// TIA Portal V17 export
// export: Created 2023-08-28T22:41:32.6164324Z, ExportSetting WithDefaults, DisplayName Totally Integrated Automation Portal, DisplayVersion V17 Update 5, DisplayName TIA Portal Openness, DisplayVersion V17 Update 5, DisplayName TIA Portal Teamcenter Gateway, DisplayVersion V17 Update 5, DisplayName TIA Portal Version Control Interface, DisplayVersion V17, DisplayName Simotion SCOUT TIA, DisplayVersion 5.4.3.0, DisplayName TIA Portal Test Suite Advanced, DisplayVersion V17 Update 1, DisplayName SIMOCODE ES, DisplayVersion V17 Update 5, DisplayName SINAMICS Startdrive Advanced, DisplayVersion V17 SP1, DisplayName SINAMICS Startdrive G130, G150, S120, S150, SINAMICS MV, S210, DisplayVersion V17 SP1, DisplayName SINAMICS Startdrive G110M, G120, G120C, G120D, G120P, G115D, DisplayVersion V17 SP1, DisplayName SIRIUS Safety ES, DisplayVersion V17 Update 5, DisplayName STEP 7 Professional, DisplayVersion V17 Update 5, DisplayName STEP 7 CFC, DisplayVersion V17 Update 1, DisplayName STEP 7 Safety, DisplayVersion V17, DisplayName WinCC Advanced, DisplayVersion V17 Update 5, DisplayName SIMATIC Visualization Architect, DisplayVersion V17 Update 5
DATA_BLOCK "S1.CABINET000.ALARM1"   // DB2200
// stored: AutoNumber true, DBAccessibleFromOPCUA true, DBAccessibleFromWebserver true, InstanceOfName BoolToUDInt_Inverted_Filtered, InstanceOfType FB
"BoolToUDInt_Inverted_Filtered "
BEGIN
END_DATA_BLOCK

DATA_BLOCK "S1.CABINET000.ALARM2"   // DB2201
// stored: AutoNumber true, DBAccessibleFromOPCUA true, DBAccessibleFromWebserver true, InstanceOfName BoolToUDInt_Inverted_Filtered, InstanceOfType FB
"BoolToUDInt_Inverted_Filtered "
BEGIN
END_DATA_BLOCK

DATA_BLOCK "S1.CABINET000.WARNING1"   // DB2202
// stored: AutoNumber true, DBAccessibleFromOPCUA true, DBAccessibleFromWebserver true, InstanceOfName BoolToUDInt_Inverted_Filtered, InstanceOfType FB
"BoolToUDInt_Inverted_Filtered "
BEGIN
END_DATA_BLOCK

DATA_BLOCK "S1.CABINET000.WARNING2"   // DB2203
// stored: AutoNumber true, DBAccessibleFromOPCUA true, DBAccessibleFromWebserver true, InstanceOfName BoolToUDInt_Inverted_Filtered, InstanceOfType FB
"BoolToUDInt_Inverted_Filtered "
BEGIN
END_DATA_BLOCK

DATA_BLOCK "S1.CABINET001.ALARM1"   // DB2204
// stored: AutoNumber true, DBAccessibleFromOPCUA true, DBAccessibleFromWebserver true, InstanceOfName BoolToUDInt_Inverted_Filtered, InstanceOfType FB
"BoolToUDInt_Inverted_Filtered "
BEGIN
END_DATA_BLOCK

DATA_BLOCK "S1.CABINET001.ALARM2"   // DB2205
// stored: AutoNumber true, DBAccessibleFromOPCUA true, DBAccessibleFromWebserver true, InstanceOfName BoolToUDInt_Inverted_Filtered, InstanceOfType FB
"BoolToUDInt_Inverted_Filtered "
BEGIN
END_DATA_BLOCK

DATA_BLOCK "S1.CABINET001.WARNING1"   // DB2206
// stored: AutoNumber true, DBAccessibleFromOPCUA true, DBAccessibleFromWebserver true, InstanceOfName BoolToUDInt_Inverted_Filtered, InstanceOfType FB
"BoolToUDInt_Inverted_Filtered "
BEGIN
END_DATA_BLOCK

DATA_BLOCK "S1.CABINET001.WARNING2"   // DB2207
// stored: AutoNumber true, DBAccessibleFromOPCUA true, DBAccessibleFromWebserver true, InstanceOfName BoolToUDInt_Inverted_Filtered, InstanceOfType FB
"BoolToUDInt_Inverted_Filtered "
BEGIN
END_DATA_BLOCK

DATA_BLOCK "S1.CABINET002.ALARM1"   // DB2208
// stored: AutoNumber true, DBAccessibleFromOPCUA true, DBAccessibleFromWebserver true, InstanceOfName BoolToUDInt_Inverted_Filtered, InstanceOfType FB
"BoolToUDInt_Inverted_Filtered "
BEGIN
END_DATA_BLOCK

DATA_BLOCK "S1.CABINET002.ALARM2"   // DB2209
// stored: AutoNumber true, DBAccessibleFromOPCUA true, DBAccessibleFromWebserver true, InstanceOfName BoolToUDInt_Inverted_Filtered, InstanceOfType FB
"BoolToUDInt_Inverted_Filtered "
BEGIN
END_DATA_BLOCK

DATA_BLOCK "S1.CABINET002.WARNING1"   // DB2210
// stored: AutoNumber true, DBAccessibleFromOPCUA true, DBAccessibleFromWebserver true, InstanceOfName BoolToUDInt_Inverted_Filtered, InstanceOfType FB
"BoolToUDInt_Inverted_Filtered "
BEGIN
END_DATA_BLOCK

DATA_BLOCK "S1.CABINET002.WARNING2"   // DB2211
// stored: AutoNumber true, DBAccessibleFromOPCUA true, DBAccessibleFromWebserver true, InstanceOfName BoolToUDInt_Inverted_Filtered, InstanceOfType FB
"BoolToUDInt_Inverted_Filtered "
BEGIN
END_DATA_BLOCK

DATA_BLOCK "S1.CABINET003.ALARM1"   // DB2212
// stored: AutoNumber true, DBAccessibleFromOPCUA true, DBAccessibleFromWebserver true, InstanceOfName BoolToUDInt_Inverted_Filtered, InstanceOfType FB
"BoolToUDInt_Inverted_Filtered "
BEGIN
END_DATA_BLOCK

DATA_BLOCK "S1.CABINET003.ALARM2"   // DB2213
// stored: AutoNumber true, DBAccessibleFromOPCUA true, DBAccessibleFromWebserver true, InstanceOfName BoolToUDInt_Inverted_Filtered, InstanceOfType FB
"BoolToUDInt_Inverted_Filtered "
BEGIN
END_DATA_BLOCK

DATA_BLOCK "S1.CABINET003.WARNING1"   // DB2214
// stored: AutoNumber true, DBAccessibleFromOPCUA true, DBAccessibleFromWebserver true, InstanceOfName BoolToUDInt_Inverted_Filtered, InstanceOfType FB
"BoolToUDInt_Inverted_Filtered "
BEGIN
END_DATA_BLOCK

DATA_BLOCK "S1.CABINET003.WARNING2"   // DB2215
// stored: AutoNumber true, DBAccessibleFromOPCUA true, DBAccessibleFromWebserver true, InstanceOfName BoolToUDInt_Inverted_Filtered, InstanceOfType FB
"BoolToUDInt_Inverted_Filtered "
BEGIN
END_DATA_BLOCK

DATA_BLOCK "S1.CABINET004.ALARM1"   // DB2216
// stored: AutoNumber true, DBAccessibleFromOPCUA true, DBAccessibleFromWebserver true, InstanceOfName BoolToUDInt_Inverted_Filtered, InstanceOfType FB
"BoolToUDInt_Inverted_Filtered "
BEGIN
END_DATA_BLOCK

DATA_BLOCK "S1.CABINET004.ALARM2"   // DB2217
// stored: AutoNumber true, DBAccessibleFromOPCUA true, DBAccessibleFromWebserver true, InstanceOfName BoolToUDInt_Inverted_Filtered, InstanceOfType FB
"BoolToUDInt_Inverted_Filtered "
BEGIN
END_DATA_BLOCK

DATA_BLOCK "S1.CABINET004.WARNING1"   // DB2218
// stored: AutoNumber true, DBAccessibleFromOPCUA true, DBAccessibleFromWebserver true, InstanceOfName BoolToUDInt_Inverted_Filtered, InstanceOfType FB
"BoolToUDInt_Inverted_Filtered "
BEGIN
END_DATA_BLOCK

DATA_BLOCK "S1.CABINET004.WARNING2"   // DB2219
// stored: AutoNumber true, DBAccessibleFromOPCUA true, DBAccessibleFromWebserver true, InstanceOfName BoolToUDInt_Inverted_Filtered, InstanceOfType FB
"BoolToUDInt_Inverted_Filtered "
BEGIN
END_DATA_BLOCK

DATA_BLOCK "S1.CABINET005.ALARM1"   // DB2220
// stored: AutoNumber true, DBAccessibleFromOPCUA true, DBAccessibleFromWebserver true, InstanceOfName BoolToUDInt_Inverted_Filtered, InstanceOfType FB
"BoolToUDInt_Inverted_Filtered "
BEGIN
END_DATA_BLOCK

DATA_BLOCK "S1.CABINET005.ALARM2"   // DB2221
// stored: AutoNumber true, DBAccessibleFromOPCUA true, DBAccessibleFromWebserver true, InstanceOfName BoolToUDInt_Inverted_Filtered, InstanceOfType FB
"BoolToUDInt_Inverted_Filtered "
BEGIN
END_DATA_BLOCK

DATA_BLOCK "S1.CABINET005.WARNING1"   // DB2222
// stored: AutoNumber true, DBAccessibleFromOPCUA true, DBAccessibleFromWebserver true, InstanceOfName BoolToUDInt_Inverted_Filtered, InstanceOfType FB
"BoolToUDInt_Inverted_Filtered "
BEGIN
END_DATA_BLOCK

DATA_BLOCK "S1.CABINET005.WARNING2"   // DB2223
// stored: AutoNumber true, DBAccessibleFromOPCUA true, DBAccessibleFromWebserver true, InstanceOfName BoolToUDInt_Inverted_Filtered, InstanceOfType FB
"BoolToUDInt_Inverted_Filtered "
BEGIN
END_DATA_BLOCK

DATA_BLOCK "S1.CABINET006.ALARM1"   // DB2224
// stored: AutoNumber true, DBAccessibleFromOPCUA true, DBAccessibleFromWebserver true, InstanceOfName BoolToUDInt_Inverted_Filtered, InstanceOfType FB
"BoolToUDInt_Inverted_Filtered "
BEGIN
END_DATA_BLOCK

DATA_BLOCK "S1.CABINET006.ALARM2"   // DB2225
// stored: AutoNumber true, DBAccessibleFromOPCUA true, DBAccessibleFromWebserver true, InstanceOfName BoolToUDInt_Inverted_Filtered, InstanceOfType FB
"BoolToUDInt_Inverted_Filtered "
BEGIN
END_DATA_BLOCK

DATA_BLOCK "S1.CABINET006.WARNING1"   // DB2226
// stored: AutoNumber true, DBAccessibleFromOPCUA true, DBAccessibleFromWebserver true, InstanceOfName BoolToUDInt_Inverted_Filtered, InstanceOfType FB
"BoolToUDInt_Inverted_Filtered "
BEGIN
END_DATA_BLOCK

DATA_BLOCK "S1.CABINET006.WARNING2"   // DB2227
// stored: AutoNumber true, DBAccessibleFromOPCUA true, DBAccessibleFromWebserver true, InstanceOfName BoolToUDInt_Inverted_Filtered, InstanceOfType FB
"BoolToUDInt_Inverted_Filtered "
BEGIN
END_DATA_BLOCK

DATA_BLOCK "S1.CABINET007.ALARM1"   // DB2228
// stored: AutoNumber true, DBAccessibleFromOPCUA true, DBAccessibleFromWebserver true, InstanceOfName BoolToUDInt_Inverted_Filtered, InstanceOfType FB
"BoolToUDInt_Inverted_Filtered "
BEGIN
END_DATA_BLOCK

DATA_BLOCK "S1.CABINET007.ALARM2"   // DB2229
// stored: AutoNumber true, DBAccessibleFromOPCUA true, DBAccessibleFromWebserver true, InstanceOfName BoolToUDInt_Inverted_Filtered, InstanceOfType FB
"BoolToUDInt_Inverted_Filtered "
BEGIN
END_DATA_BLOCK

DATA_BLOCK "S1.CABINET007.WARNING1"   // DB2230
// stored: AutoNumber true, DBAccessibleFromOPCUA true, DBAccessibleFromWebserver true, InstanceOfName BoolToUDInt_Inverted_Filtered, InstanceOfType FB
"BoolToUDInt_Inverted_Filtered "
BEGIN
END_DATA_BLOCK

DATA_BLOCK "S1.CABINET007.WARNING2"   // DB2231
// stored: AutoNumber true, DBAccessibleFromOPCUA true, DBAccessibleFromWebserver true, InstanceOfName BoolToUDInt_Inverted_Filtered, InstanceOfType FB
"BoolToUDInt_Inverted_Filtered "
BEGIN
END_DATA_BLOCK

DATA_BLOCK "S1.CABINET008.ALARM1"   // DB2232
// stored: AutoNumber true, DBAccessibleFromOPCUA true, DBAccessibleFromWebserver true, InstanceOfName BoolToUDInt_Inverted_Filtered, InstanceOfType FB
"BoolToUDInt_Inverted_Filtered "
BEGIN
END_DATA_BLOCK

DATA_BLOCK "S1.CABINET008.ALARM2"   // DB2233
// stored: AutoNumber true, DBAccessibleFromOPCUA true, DBAccessibleFromWebserver true, InstanceOfName BoolToUDInt_Inverted_Filtered, InstanceOfType FB
"BoolToUDInt_Inverted_Filtered "
BEGIN
END_DATA_BLOCK

DATA_BLOCK "S1.CABINET008.WARNING1"   // DB2234
// stored: AutoNumber true, DBAccessibleFromOPCUA true, DBAccessibleFromWebserver true, InstanceOfName BoolToUDInt_Inverted_Filtered, InstanceOfType FB
"BoolToUDInt_Inverted_Filtered "
BEGIN
END_DATA_BLOCK

DATA_BLOCK "S1.CABINET008.WARNING2"   // DB2235
// stored: AutoNumber true, DBAccessibleFromOPCUA true, DBAccessibleFromWebserver true, InstanceOfName BoolToUDInt_Inverted_Filtered, InstanceOfType FB
"BoolToUDInt_Inverted_Filtered "
BEGIN
END_DATA_BLOCK

DATA_BLOCK "S1.CABINET009.ALARM1"   // DB2236
// stored: AutoNumber true, DBAccessibleFromOPCUA true, DBAccessibleFromWebserver true, InstanceOfName BoolToUDInt_Inverted_Filtered, InstanceOfType FB
"BoolToUDInt_Inverted_Filtered "
BEGIN
END_DATA_BLOCK

DATA_BLOCK "S1.CABINET009.ALARM2"   // DB2237
// stored: AutoNumber true, DBAccessibleFromOPCUA true, DBAccessibleFromWebserver true, InstanceOfName BoolToUDInt_Inverted_Filtered, InstanceOfType FB
"BoolToUDInt_Inverted_Filtered "
BEGIN
END_DATA_BLOCK

DATA_BLOCK "S1.CABINET009.WARNING1"   // DB2238
// stored: AutoNumber true, DBAccessibleFromOPCUA true, DBAccessibleFromWebserver true, InstanceOfName BoolToUDInt_Inverted_Filtered, InstanceOfType FB
"BoolToUDInt_Inverted_Filtered "
BEGIN
END_DATA_BLOCK

DATA_BLOCK "S1.CABINET009.WARNING2"   // DB2239
// stored: AutoNumber true, DBAccessibleFromOPCUA true, DBAccessibleFromWebserver true, InstanceOfName BoolToUDInt_Inverted_Filtered, InstanceOfType FB
"BoolToUDInt_Inverted_Filtered "
BEGIN
END_DATA_BLOCK

DATA_BLOCK "S1.CABINET010.ALARM1"   // DB2240
// stored: AutoNumber true, DBAccessibleFromOPCUA true, DBAccessibleFromWebserver true, InstanceOfName BoolToUDInt_Inverted_Filtered, InstanceOfType FB
"BoolToUDInt_Inverted_Filtered "
BEGIN
END_DATA_BLOCK

DATA_BLOCK "S1.CABINET010.ALARM2"   // DB2241
// stored: AutoNumber true, DBAccessibleFromOPCUA true, DBAccessibleFromWebserver true, InstanceOfName BoolToUDInt_Inverted_Filtered, InstanceOfType FB
"BoolToUDInt_Inverted_Filtered "
BEGIN
END_DATA_BLOCK

DATA_BLOCK "S1.CABINET010.WARNING1"   // DB2242
// stored: AutoNumber true, DBAccessibleFromOPCUA true, DBAccessibleFromWebserver true, InstanceOfName BoolToUDInt_Inverted_Filtered, InstanceOfType FB
"BoolToUDInt_Inverted_Filtered "
BEGIN
END_DATA_BLOCK

DATA_BLOCK "S1.CABINET010.WARNING2"   // DB2243
// stored: AutoNumber true, DBAccessibleFromOPCUA true, DBAccessibleFromWebserver true, InstanceOfName BoolToUDInt_Inverted_Filtered, InstanceOfType FB
"BoolToUDInt_Inverted_Filtered "
BEGIN
END_DATA_BLOCK

DATA_BLOCK "S1.CABINET011.ALARM1"   // DB2244
// stored: AutoNumber true, DBAccessibleFromOPCUA true, DBAccessibleFromWebserver true, InstanceOfName BoolToUDInt_Inverted_Filtered, InstanceOfType FB
"BoolToUDInt_Inverted_Filtered "
BEGIN
END_DATA_BLOCK

DATA_BLOCK "S1.CABINET011.ALARM2"   // DB2245
// stored: AutoNumber true, DBAccessibleFromOPCUA true, DBAccessibleFromWebserver true, InstanceOfName BoolToUDInt_Inverted_Filtered, InstanceOfType FB
"BoolToUDInt_Inverted_Filtered "
BEGIN
END_DATA_BLOCK

DATA_BLOCK "S1.CABINET011.WARNING1"   // DB2246
// stored: AutoNumber true, DBAccessibleFromOPCUA true, DBAccessibleFromWebserver true, InstanceOfName BoolToUDInt_Inverted_Filtered, InstanceOfType FB
"BoolToUDInt_Inverted_Filtered "
BEGIN
END_DATA_BLOCK

DATA_BLOCK "S1.CABINET011.WARNING2"   // DB2247
// stored: AutoNumber true, DBAccessibleFromOPCUA true, DBAccessibleFromWebserver true, InstanceOfName BoolToUDInt_Inverted_Filtered, InstanceOfType FB
"BoolToUDInt_Inverted_Filtered "
BEGIN
END_DATA_BLOCK

DATA_BLOCK "S1.CABINET012.ALARM1"   // DB2248
// stored: AutoNumber true, DBAccessibleFromOPCUA true, DBAccessibleFromWebserver true, InstanceOfName BoolToUDInt_Inverted_Filtered, InstanceOfType FB
"BoolToUDInt_Inverted_Filtered "
BEGIN
END_DATA_BLOCK

DATA_BLOCK "S1.CABINET012.ALARM2"   // DB2249
// stored: AutoNumber true, DBAccessibleFromOPCUA true, DBAccessibleFromWebserver true, InstanceOfName BoolToUDInt_Inverted_Filtered, InstanceOfType FB
"BoolToUDInt_Inverted_Filtered "
BEGIN
END_DATA_BLOCK

DATA_BLOCK "S1.CABINET012.WARNING1"   // DB2250
// stored: AutoNumber true, DBAccessibleFromOPCUA true, DBAccessibleFromWebserver true, InstanceOfName BoolToUDInt_Inverted_Filtered, InstanceOfType FB
"BoolToUDInt_Inverted_Filtered "
BEGIN
END_DATA_BLOCK

DATA_BLOCK "S1.CABINET012.WARNING2"   // DB2251
// stored: AutoNumber true, DBAccessibleFromOPCUA true, DBAccessibleFromWebserver true, InstanceOfName BoolToUDInt_Inverted_Filtered, InstanceOfType FB
"BoolToUDInt_Inverted_Filtered "
BEGIN
END_DATA_BLOCK

DATA_BLOCK "S1.CABINET013.ALARM1"   // DB2252
// stored: AutoNumber true, DBAccessibleFromOPCUA true, DBAccessibleFromWebserver true, InstanceOfName BoolToUDInt_Inverted_Filtered, InstanceOfType FB
"BoolToUDInt_Inverted_Filtered "
BEGIN
END_DATA_BLOCK

DATA_BLOCK "S1.CABINET013.ALARM2"   // DB2253
// stored: AutoNumber true, DBAccessibleFromOPCUA true, DBAccessibleFromWebserver true, InstanceOfName BoolToUDInt_Inverted_Filtered, InstanceOfType FB
"BoolToUDInt_Inverted_Filtered "
BEGIN
END_DATA_BLOCK

DATA_BLOCK "S1.CABINET013.WARNING1"   // DB2254
// stored: AutoNumber true, DBAccessibleFromOPCUA true, DBAccessibleFromWebserver true, InstanceOfName BoolToUDInt_Inverted_Filtered, InstanceOfType FB
"BoolToUDInt_Inverted_Filtered "
BEGIN
END_DATA_BLOCK

DATA_BLOCK "S1.CABINET013.WARNING2"   // DB2255
// stored: AutoNumber true, DBAccessibleFromOPCUA true, DBAccessibleFromWebserver true, InstanceOfName BoolToUDInt_Inverted_Filtered, InstanceOfType FB
"BoolToUDInt_Inverted_Filtered "
BEGIN
END_DATA_BLOCK

DATA_BLOCK "S1.CABINET014.ALARM1"   // DB2256
// stored: AutoNumber true, DBAccessibleFromOPCUA true, DBAccessibleFromWebserver true, InstanceOfName BoolToUDInt_Inverted_Filtered, InstanceOfType FB
"BoolToUDInt_Inverted_Filtered "
BEGIN
END_DATA_BLOCK

DATA_BLOCK "S1.CABINET014.ALARM2"   // DB2257
// stored: AutoNumber true, DBAccessibleFromOPCUA true, DBAccessibleFromWebserver true, InstanceOfName BoolToUDInt_Inverted_Filtered, InstanceOfType FB
"BoolToUDInt_Inverted_Filtered "
BEGIN
END_DATA_BLOCK

DATA_BLOCK "S1.CABINET014.WARNING1"   // DB2258
// stored: AutoNumber true, DBAccessibleFromOPCUA true, DBAccessibleFromWebserver true, InstanceOfName BoolToUDInt_Inverted_Filtered, InstanceOfType FB
"BoolToUDInt_Inverted_Filtered "
BEGIN
END_DATA_BLOCK

DATA_BLOCK "S1.CABINET014.WARNING2"   // DB2259
// stored: AutoNumber true, DBAccessibleFromOPCUA true, DBAccessibleFromWebserver true, InstanceOfName BoolToUDInt_Inverted_Filtered, InstanceOfType FB
"BoolToUDInt_Inverted_Filtered "
BEGIN
END_DATA_BLOCK

DATA_BLOCK "S1.CABINET015.ALARM1"   // DB2260
// stored: AutoNumber true, DBAccessibleFromOPCUA true, DBAccessibleFromWebserver true, InstanceOfName BoolToUDInt_Inverted_Filtered, InstanceOfType FB
"BoolToUDInt_Inverted_Filtered "
BEGIN
END_DATA_BLOCK

DATA_BLOCK "S1.CABINET015.ALARM2"   // DB2261
// stored: AutoNumber true, DBAccessibleFromOPCUA true, DBAccessibleFromWebserver true, InstanceOfName BoolToUDInt_Inverted_Filtered, InstanceOfType FB
"BoolToUDInt_Inverted_Filtered "
BEGIN
END_DATA_BLOCK

DATA_BLOCK "S1.CABINET015.WARNING1"   // DB2262
// stored: AutoNumber true, DBAccessibleFromOPCUA true, DBAccessibleFromWebserver true, InstanceOfName BoolToUDInt_Inverted_Filtered, InstanceOfType FB
"BoolToUDInt_Inverted_Filtered "
BEGIN
END_DATA_BLOCK

DATA_BLOCK "S1.CABINET015.WARNING2"   // DB2263
// stored: AutoNumber true, DBAccessibleFromOPCUA true, DBAccessibleFromWebserver true, InstanceOfName BoolToUDInt_Inverted_Filtered, InstanceOfType FB
"BoolToUDInt_Inverted_Filtered "
BEGIN
END_DATA_BLOCK

DATA_BLOCK "S1.CABINET016.ALARM1"   // DB2264
// stored: AutoNumber true, DBAccessibleFromOPCUA true, DBAccessibleFromWebserver true, InstanceOfName BoolToUDInt_Inverted_Filtered, InstanceOfType FB
"BoolToUDInt_Inverted_Filtered "
BEGIN
END_DATA_BLOCK

DATA_BLOCK "S1.CABINET016.ALARM2"   // DB2265
// stored: AutoNumber true, DBAccessibleFromOPCUA true, DBAccessibleFromWebserver true, InstanceOfName BoolToUDInt_Inverted_Filtered, InstanceOfType FB
"BoolToUDInt_Inverted_Filtered "
BEGIN
END_DATA_BLOCK

DATA_BLOCK "S1.CABINET016.WARNING1"   // DB2266
// stored: AutoNumber true, DBAccessibleFromOPCUA true, DBAccessibleFromWebserver true, InstanceOfName BoolToUDInt_Inverted_Filtered, InstanceOfType FB
"BoolToUDInt_Inverted_Filtered "
BEGIN
END_DATA_BLOCK

DATA_BLOCK "S1.CABINET016.WARNING2"   // DB2267
// stored: AutoNumber true, DBAccessibleFromOPCUA true, DBAccessibleFromWebserver true, InstanceOfName BoolToUDInt_Inverted_Filtered, InstanceOfType FB
"BoolToUDInt_Inverted_Filtered "
BEGIN
END_DATA_BLOCK

DATA_BLOCK "S1.CABINET017.ALARM1"   // DB2268
// stored: AutoNumber true, DBAccessibleFromOPCUA true, DBAccessibleFromWebserver true, InstanceOfName BoolToUDInt_Inverted_Filtered, InstanceOfType FB
"BoolToUDInt_Inverted_Filtered "
BEGIN
END_DATA_BLOCK

DATA_BLOCK "S1.CABINET017.ALARM2"   // DB2269
// stored: AutoNumber true, DBAccessibleFromOPCUA true, DBAccessibleFromWebserver true, InstanceOfName BoolToUDInt_Inverted_Filtered, InstanceOfType FB
"BoolToUDInt_Inverted_Filtered "
BEGIN
END_DATA_BLOCK

DATA_BLOCK "S1.CABINET017.WARNING1"   // DB2270
// stored: AutoNumber true, DBAccessibleFromOPCUA true, DBAccessibleFromWebserver true, InstanceOfName BoolToUDInt_Inverted_Filtered, InstanceOfType FB
"BoolToUDInt_Inverted_Filtered "
BEGIN
END_DATA_BLOCK

DATA_BLOCK "S1.CABINET017.WARNING2"   // DB2271
// stored: AutoNumber true, DBAccessibleFromOPCUA true, DBAccessibleFromWebserver true, InstanceOfName BoolToUDInt_Inverted_Filtered, InstanceOfType FB
"BoolToUDInt_Inverted_Filtered "
BEGIN
END_DATA_BLOCK

DATA_BLOCK "S1.CABINET018.ALARM1"   // DB2272
// stored: AutoNumber true, DBAccessibleFromOPCUA true, DBAccessibleFromWebserver true, InstanceOfName BoolToUDInt_Inverted_Filtered, InstanceOfType FB
"BoolToUDInt_Inverted_Filtered "
BEGIN
END_DATA_BLOCK

DATA_BLOCK "S1.CABINET018.ALARM2"   // DB2273
// stored: AutoNumber true, DBAccessibleFromOPCUA true, DBAccessibleFromWebserver true, InstanceOfName BoolToUDInt_Inverted_Filtered, InstanceOfType FB
"BoolToUDInt_Inverted_Filtered "
BEGIN
END_DATA_BLOCK

DATA_BLOCK "S1.CABINET018.WARNING1"   // DB2274
// stored: AutoNumber true, DBAccessibleFromOPCUA true, DBAccessibleFromWebserver true, InstanceOfName BoolToUDInt_Inverted_Filtered, InstanceOfType FB
"BoolToUDInt_Inverted_Filtered "
BEGIN
END_DATA_BLOCK

DATA_BLOCK "S1.CABINET018.WARNING2"   // DB2275
// stored: AutoNumber true, DBAccessibleFromOPCUA true, DBAccessibleFromWebserver true, InstanceOfName BoolToUDInt_Inverted_Filtered, InstanceOfType FB
"BoolToUDInt_Inverted_Filtered "
BEGIN
END_DATA_BLOCK

DATA_BLOCK "S1.CABINET019.ALARM1"   // DB2276
// stored: AutoNumber true, DBAccessibleFromOPCUA true, DBAccessibleFromWebserver true, InstanceOfName BoolToUDInt_Inverted_Filtered, InstanceOfType FB
"BoolToUDInt_Inverted_Filtered "
BEGIN
END_DATA_BLOCK

DATA_BLOCK "S1.CABINET019.ALARM2"   // DB2277
// stored: AutoNumber true, DBAccessibleFromOPCUA true, DBAccessibleFromWebserver true, InstanceOfName BoolToUDInt_Inverted_Filtered, InstanceOfType FB
"BoolToUDInt_Inverted_Filtered "
BEGIN
END_DATA_BLOCK

DATA_BLOCK "S1.CABINET019.WARNING1"   // DB2278
// stored: AutoNumber true, DBAccessibleFromOPCUA true, DBAccessibleFromWebserver true, InstanceOfName BoolToUDInt_Inverted_Filtered, InstanceOfType FB
"BoolToUDInt_Inverted_Filtered "
BEGIN
END_DATA_BLOCK

DATA_BLOCK "S1.CABINET019.WARNING2"   // DB2279
// stored: AutoNumber true, DBAccessibleFromOPCUA true, DBAccessibleFromWebserver true, InstanceOfName BoolToUDInt_Inverted_Filtered, InstanceOfType FB
"BoolToUDInt_Inverted_Filtered "
BEGIN
END_DATA_BLOCK

DATA_BLOCK "S1.CABINET020.ALARM1"   // DB2280
// stored: AutoNumber true, DBAccessibleFromOPCUA true, DBAccessibleFromWebserver true, InstanceOfName BoolToUDInt_Inverted_Filtered, InstanceOfType FB
"BoolToUDInt_Inverted_Filtered "
BEGIN
END_DATA_BLOCK

DATA_BLOCK "S1.CABINET020.ALARM2"   // DB2281
// stored: AutoNumber true, DBAccessibleFromOPCUA true, DBAccessibleFromWebserver true, InstanceOfName BoolToUDInt_Inverted_Filtered, InstanceOfType FB
"BoolToUDInt_Inverted_Filtered "
BEGIN
END_DATA_BLOCK

DATA_BLOCK "S1.CABINET020.WARNING1"   // DB2282
// stored: AutoNumber true, DBAccessibleFromOPCUA true, DBAccessibleFromWebserver true, InstanceOfName BoolToUDInt_Inverted_Filtered, InstanceOfType FB
"BoolToUDInt_Inverted_Filtered "
BEGIN
END_DATA_BLOCK

DATA_BLOCK "S1.CABINET020.WARNING2"   // DB2283
// stored: AutoNumber true, DBAccessibleFromOPCUA true, DBAccessibleFromWebserver true, InstanceOfName BoolToUDInt_Inverted_Filtered, InstanceOfType FB
"BoolToUDInt_Inverted_Filtered "
BEGIN
END_DATA_BLOCK

DATA_BLOCK "S1.CABINET021.ALARM1"   // DB2284
// stored: AutoNumber true, DBAccessibleFromOPCUA true, DBAccessibleFromWebserver true, InstanceOfName BoolToUDInt_Inverted_Filtered, InstanceOfType FB
"BoolToUDInt_Inverted_Filtered "
BEGIN
END_DATA_BLOCK

DATA_BLOCK "S1.CABINET021.ALARM2"   // DB2285
// stored: AutoNumber true, DBAccessibleFromOPCUA true, DBAccessibleFromWebserver true, InstanceOfName BoolToUDInt_Inverted_Filtered, InstanceOfType FB
"BoolToUDInt_Inverted_Filtered "
BEGIN
END_DATA_BLOCK

DATA_BLOCK "S1.CABINET021.WARNING1"   // DB2286
// stored: AutoNumber true, DBAccessibleFromOPCUA true, DBAccessibleFromWebserver true, InstanceOfName BoolToUDInt_Inverted_Filtered, InstanceOfType FB
"BoolToUDInt_Inverted_Filtered "
BEGIN
END_DATA_BLOCK

DATA_BLOCK "S1.CABINET021.WARNING2"   // DB2287
// stored: AutoNumber true, DBAccessibleFromOPCUA true, DBAccessibleFromWebserver true, InstanceOfName BoolToUDInt_Inverted_Filtered, InstanceOfType FB
"BoolToUDInt_Inverted_Filtered "
BEGIN
END_DATA_BLOCK

DATA_BLOCK "S1.CABINET022.ALARM1"   // DB2288
// stored: AutoNumber true, DBAccessibleFromOPCUA true, DBAccessibleFromWebserver true, InstanceOfName BoolToUDInt_Inverted_Filtered, InstanceOfType FB
"BoolToUDInt_Inverted_Filtered "
BEGIN
END_DATA_BLOCK

DATA_BLOCK "S1.CABINET022.ALARM2"   // DB2289
// stored: AutoNumber true, DBAccessibleFromOPCUA true, DBAccessibleFromWebserver true, InstanceOfName BoolToUDInt_Inverted_Filtered, InstanceOfType FB
"BoolToUDInt_Inverted_Filtered "
BEGIN
END_DATA_BLOCK

DATA_BLOCK "S1.CABINET022.WARNING1"   // DB2290
// stored: AutoNumber true, DBAccessibleFromOPCUA true, DBAccessibleFromWebserver true, InstanceOfName BoolToUDInt_Inverted_Filtered, InstanceOfType FB
"BoolToUDInt_Inverted_Filtered "
BEGIN
END_DATA_BLOCK

DATA_BLOCK "S1.CABINET022.WARNING2"   // DB2291
// stored: AutoNumber true, DBAccessibleFromOPCUA true, DBAccessibleFromWebserver true, InstanceOfName BoolToUDInt_Inverted_Filtered, InstanceOfType FB
"BoolToUDInt_Inverted_Filtered "
BEGIN
END_DATA_BLOCK

DATA_BLOCK "S1.CABINET023.ALARM1"   // DB2292
// stored: AutoNumber true, DBAccessibleFromOPCUA true, DBAccessibleFromWebserver true, InstanceOfName BoolToUDInt_Inverted_Filtered, InstanceOfType FB
"BoolToUDInt_Inverted_Filtered "
BEGIN
END_DATA_BLOCK

DATA_BLOCK "S1.CABINET023.ALARM2"   // DB2293
// stored: AutoNumber true, DBAccessibleFromOPCUA true, DBAccessibleFromWebserver true, InstanceOfName BoolToUDInt_Inverted_Filtered, InstanceOfType FB
"BoolToUDInt_Inverted_Filtered "
BEGIN
END_DATA_BLOCK

DATA_BLOCK "S1.CABINET023.WARNING1"   // DB2294
// stored: AutoNumber true, DBAccessibleFromOPCUA true, DBAccessibleFromWebserver true, InstanceOfName BoolToUDInt_Inverted_Filtered, InstanceOfType FB
"BoolToUDInt_Inverted_Filtered "
BEGIN
END_DATA_BLOCK

DATA_BLOCK "S1.CABINET023.WARNING2"   // DB2295
// stored: AutoNumber true, DBAccessibleFromOPCUA true, DBAccessibleFromWebserver true, InstanceOfName BoolToUDInt_Inverted_Filtered, InstanceOfType FB
"BoolToUDInt_Inverted_Filtered "
BEGIN
END_DATA_BLOCK

DATA_BLOCK "S1.CABINET024.ALARM1"   // DB2296
// stored: AutoNumber true, DBAccessibleFromOPCUA true, DBAccessibleFromWebserver true, InstanceOfName BoolToUDInt_Inverted_Filtered, InstanceOfType FB
"BoolToUDInt_Inverted_Filtered "
BEGIN
END_DATA_BLOCK

DATA_BLOCK "S1.CABINET024.ALARM2"   // DB2297
// stored: AutoNumber true, DBAccessibleFromOPCUA true, DBAccessibleFromWebserver true, InstanceOfName BoolToUDInt_Inverted_Filtered, InstanceOfType FB
"BoolToUDInt_Inverted_Filtered "
BEGIN
END_DATA_BLOCK

DATA_BLOCK "S1.CABINET024.WARNING1"   // DB2298
// stored: AutoNumber true, DBAccessibleFromOPCUA true, DBAccessibleFromWebserver true, InstanceOfName BoolToUDInt_Inverted_Filtered, InstanceOfType FB
"BoolToUDInt_Inverted_Filtered "
BEGIN
END_DATA_BLOCK

DATA_BLOCK "S1.CABINET024.WARNING2"   // DB2299
// stored: AutoNumber true, DBAccessibleFromOPCUA true, DBAccessibleFromWebserver true, InstanceOfName BoolToUDInt_Inverted_Filtered, InstanceOfType FB
"BoolToUDInt_Inverted_Filtered "
BEGIN
END_DATA_BLOCK

DATA_BLOCK "S1.CABINET025.ALARM1"   // DB2300
// stored: AutoNumber true, DBAccessibleFromOPCUA true, DBAccessibleFromWebserver true, InstanceOfName BoolToUDInt_Inverted_Filtered, InstanceOfType FB
"BoolToUDInt_Inverted_Filtered "
BEGIN
END_DATA_BLOCK

DATA_BLOCK "S1.CABINET025.ALARM2"   // DB2301
// stored: AutoNumber true, DBAccessibleFromOPCUA true, DBAccessibleFromWebserver true, InstanceOfName BoolToUDInt_Inverted_Filtered, InstanceOfType FB
"BoolToUDInt_Inverted_Filtered "
BEGIN
END_DATA_BLOCK

DATA_BLOCK "S1.CABINET025.WARNING1"   // DB2302
// stored: AutoNumber true, DBAccessibleFromOPCUA true, DBAccessibleFromWebserver true, InstanceOfName BoolToUDInt_Inverted_Filtered, InstanceOfType FB
"BoolToUDInt_Inverted_Filtered "
BEGIN
END_DATA_BLOCK

DATA_BLOCK "S1.CABINET025.WARNING2"   // DB2303
// stored: AutoNumber true, DBAccessibleFromOPCUA true, DBAccessibleFromWebserver true, InstanceOfName BoolToUDInt_Inverted_Filtered, InstanceOfType FB
"BoolToUDInt_Inverted_Filtered "
BEGIN
END_DATA_BLOCK

DATA_BLOCK "S1.CABINET026.ALARM1"   // DB2304
// stored: AutoNumber true, DBAccessibleFromOPCUA true, DBAccessibleFromWebserver true, InstanceOfName BoolToUDInt_Inverted_Filtered, InstanceOfType FB
"BoolToUDInt_Inverted_Filtered "
BEGIN
END_DATA_BLOCK

DATA_BLOCK "S1.CABINET026.ALARM2"   // DB2305
// stored: AutoNumber true, DBAccessibleFromOPCUA true, DBAccessibleFromWebserver true, InstanceOfName BoolToUDInt_Inverted_Filtered, InstanceOfType FB
"BoolToUDInt_Inverted_Filtered "
BEGIN
END_DATA_BLOCK

DATA_BLOCK "S1.CABINET026.WARNING1"   // DB2306
// stored: AutoNumber true, DBAccessibleFromOPCUA true, DBAccessibleFromWebserver true, InstanceOfName BoolToUDInt_Inverted_Filtered, InstanceOfType FB
"BoolToUDInt_Inverted_Filtered "
BEGIN
END_DATA_BLOCK

DATA_BLOCK "S1.CABINET026.WARNING2"   // DB2307
// stored: AutoNumber true, DBAccessibleFromOPCUA true, DBAccessibleFromWebserver true, InstanceOfName BoolToUDInt_Inverted_Filtered, InstanceOfType FB
"BoolToUDInt_Inverted_Filtered "
BEGIN
END_DATA_BLOCK

DATA_BLOCK "S1.CABINET027.ALARM1"   // DB2308
// stored: AutoNumber true, DBAccessibleFromOPCUA true, DBAccessibleFromWebserver true, InstanceOfName BoolToUDInt_Inverted_Filtered, InstanceOfType FB
"BoolToUDInt_Inverted_Filtered "
BEGIN
END_DATA_BLOCK

DATA_BLOCK "S1.CABINET027.ALARM2"   // DB2309
// stored: AutoNumber true, DBAccessibleFromOPCUA true, DBAccessibleFromWebserver true, InstanceOfName BoolToUDInt_Inverted_Filtered, InstanceOfType FB
"BoolToUDInt_Inverted_Filtered "
BEGIN
END_DATA_BLOCK

DATA_BLOCK "S1.CABINET027.WARNING1"   // DB2310
// stored: AutoNumber true, DBAccessibleFromOPCUA true, DBAccessibleFromWebserver true, InstanceOfName BoolToUDInt_Inverted_Filtered, InstanceOfType FB
"BoolToUDInt_Inverted_Filtered "
BEGIN
END_DATA_BLOCK

DATA_BLOCK "S1.CABINET027.WARNING2"   // DB2311
// stored: AutoNumber true, DBAccessibleFromOPCUA true, DBAccessibleFromWebserver true, InstanceOfName BoolToUDInt_Inverted_Filtered, InstanceOfType FB
"BoolToUDInt_Inverted_Filtered "
BEGIN
END_DATA_BLOCK

DATA_BLOCK "S1.CABINET028.ALARM1"   // DB2312
// stored: AutoNumber true, DBAccessibleFromOPCUA true, DBAccessibleFromWebserver true, InstanceOfName BoolToUDInt_Inverted_Filtered, InstanceOfType FB
"BoolToUDInt_Inverted_Filtered "
BEGIN
END_DATA_BLOCK

DATA_BLOCK "S1.CABINET028.ALARM2"   // DB2313
// stored: AutoNumber true, DBAccessibleFromOPCUA true, DBAccessibleFromWebserver true, InstanceOfName BoolToUDInt_Inverted_Filtered, InstanceOfType FB
"BoolToUDInt_Inverted_Filtered "
BEGIN
END_DATA_BLOCK

DATA_BLOCK "S1.CABINET028.WARNING1"   // DB2314
// stored: AutoNumber true, DBAccessibleFromOPCUA true, DBAccessibleFromWebserver true, InstanceOfName BoolToUDInt_Inverted_Filtered, InstanceOfType FB
"BoolToUDInt_Inverted_Filtered "
BEGIN
END_DATA_BLOCK

DATA_BLOCK "S1.CABINET028.WARNING2"   // DB2315
// stored: AutoNumber true, DBAccessibleFromOPCUA true, DBAccessibleFromWebserver true, InstanceOfName BoolToUDInt_Inverted_Filtered, InstanceOfType FB
"BoolToUDInt_Inverted_Filtered "
BEGIN
END_DATA_BLOCK

DATA_BLOCK "S1.CABINET029.ALARM1"   // DB2316
// stored: AutoNumber true, DBAccessibleFromOPCUA true, DBAccessibleFromWebserver true, InstanceOfName BoolToUDInt_Inverted_Filtered, InstanceOfType FB
"BoolToUDInt_Inverted_Filtered "
BEGIN
END_DATA_BLOCK

DATA_BLOCK "S1.CABINET029.ALARM2"   // DB2317
// stored: AutoNumber true, DBAccessibleFromOPCUA true, DBAccessibleFromWebserver true, InstanceOfName BoolToUDInt_Inverted_Filtered, InstanceOfType FB
"BoolToUDInt_Inverted_Filtered "
BEGIN
END_DATA_BLOCK

DATA_BLOCK "S1.CABINET029.WARNING1"   // DB2318
// stored: AutoNumber true, DBAccessibleFromOPCUA true, DBAccessibleFromWebserver true, InstanceOfName BoolToUDInt_Inverted_Filtered, InstanceOfType FB
"BoolToUDInt_Inverted_Filtered "
BEGIN
END_DATA_BLOCK

DATA_BLOCK "S1.CABINET029.WARNING2"   // DB2319
// stored: AutoNumber true, DBAccessibleFromOPCUA true, DBAccessibleFromWebserver true, InstanceOfName BoolToUDInt_Inverted_Filtered, InstanceOfType FB
"BoolToUDInt_Inverted_Filtered "
BEGIN
END_DATA_BLOCK

DATA_BLOCK "S1.CABINET030.ALARM1"   // DB2320
// stored: AutoNumber true, DBAccessibleFromOPCUA true, DBAccessibleFromWebserver true, InstanceOfName BoolToUDInt_Inverted_Filtered, InstanceOfType FB
"BoolToUDInt_Inverted_Filtered "
BEGIN
END_DATA_BLOCK

DATA_BLOCK "S1.CABINET030.ALARM2"   // DB2321
// stored: AutoNumber true, DBAccessibleFromOPCUA true, DBAccessibleFromWebserver true, InstanceOfName BoolToUDInt_Inverted_Filtered, InstanceOfType FB
"BoolToUDInt_Inverted_Filtered "
BEGIN
END_DATA_BLOCK

DATA_BLOCK "S1.CABINET030.WARNING1"   // DB2322
// stored: AutoNumber true, DBAccessibleFromOPCUA true, DBAccessibleFromWebserver true, InstanceOfName BoolToUDInt_Inverted_Filtered, InstanceOfType FB
"BoolToUDInt_Inverted_Filtered "
BEGIN
END_DATA_BLOCK

DATA_BLOCK "S1.CABINET030.WARNING2"   // DB2323
// stored: AutoNumber true, DBAccessibleFromOPCUA true, DBAccessibleFromWebserver true, InstanceOfName BoolToUDInt_Inverted_Filtered, InstanceOfType FB
"BoolToUDInt_Inverted_Filtered "
BEGIN
END_DATA_BLOCK

DATA_BLOCK "S1.CABINET031.ALARM1"   // DB2324
// stored: AutoNumber true, DBAccessibleFromOPCUA true, DBAccessibleFromWebserver true, InstanceOfName BoolToUDInt_Inverted_Filtered, InstanceOfType FB
"BoolToUDInt_Inverted_Filtered "
BEGIN
END_DATA_BLOCK

DATA_BLOCK "S1.CABINET031.ALARM2"   // DB2325
// stored: AutoNumber true, DBAccessibleFromOPCUA true, DBAccessibleFromWebserver true, InstanceOfName BoolToUDInt_Inverted_Filtered, InstanceOfType FB
"BoolToUDInt_Inverted_Filtered "
BEGIN
END_DATA_BLOCK

DATA_BLOCK "S1.CABINET031.WARNING1"   // DB2326
// stored: AutoNumber true, DBAccessibleFromOPCUA true, DBAccessibleFromWebserver true, InstanceOfName BoolToUDInt_Inverted_Filtered, InstanceOfType FB
"BoolToUDInt_Inverted_Filtered "
BEGIN
END_DATA_BLOCK

DATA_BLOCK "S1.CABINET031.WARNING2"   // DB2327
// stored: AutoNumber true, DBAccessibleFromOPCUA true, DBAccessibleFromWebserver true, InstanceOfName BoolToUDInt_Inverted_Filtered, InstanceOfType FB
"BoolToUDInt_Inverted_Filtered "
BEGIN
END_DATA_BLOCK

DATA_BLOCK "S1.CABINET032.ALARM1"   // DB2328
// stored: AutoNumber true, DBAccessibleFromOPCUA true, DBAccessibleFromWebserver true, InstanceOfName BoolToUDInt_Inverted_Filtered, InstanceOfType FB
"BoolToUDInt_Inverted_Filtered "
BEGIN
END_DATA_BLOCK

DATA_BLOCK "S1.CABINET032.ALARM2"   // DB2329
// stored: AutoNumber true, DBAccessibleFromOPCUA true, DBAccessibleFromWebserver true, InstanceOfName BoolToUDInt_Inverted_Filtered, InstanceOfType FB
"BoolToUDInt_Inverted_Filtered "
BEGIN
END_DATA_BLOCK

DATA_BLOCK "S1.CABINET032.WARNING1"   // DB2330
// stored: AutoNumber true, DBAccessibleFromOPCUA true, DBAccessibleFromWebserver true, InstanceOfName BoolToUDInt_Inverted_Filtered, InstanceOfType FB
"BoolToUDInt_Inverted_Filtered "
BEGIN
END_DATA_BLOCK

DATA_BLOCK "S1.CABINET032.WARNING2"   // DB2331
// stored: AutoNumber true, DBAccessibleFromOPCUA true, DBAccessibleFromWebserver true, InstanceOfName BoolToUDInt_Inverted_Filtered, InstanceOfType FB
"BoolToUDInt_Inverted_Filtered "
BEGIN
END_DATA_BLOCK

DATA_BLOCK "S1.CABINET033.ALARM1"   // DB2332
// stored: AutoNumber true, DBAccessibleFromOPCUA true, DBAccessibleFromWebserver true, InstanceOfName BoolToUDInt_Inverted_Filtered, InstanceOfType FB
"BoolToUDInt_Inverted_Filtered "
BEGIN
END_DATA_BLOCK

DATA_BLOCK "S1.CABINET033.ALARM2"   // DB2333
// stored: AutoNumber true, DBAccessibleFromOPCUA true, DBAccessibleFromWebserver true, InstanceOfName BoolToUDInt_Inverted_Filtered, InstanceOfType FB
"BoolToUDInt_Inverted_Filtered "
BEGIN
END_DATA_BLOCK

DATA_BLOCK "S1.CABINET033.WARNING1"   // DB2334
// stored: AutoNumber true, DBAccessibleFromOPCUA true, DBAccessibleFromWebserver true, InstanceOfName BoolToUDInt_Inverted_Filtered, InstanceOfType FB
"BoolToUDInt_Inverted_Filtered "
BEGIN
END_DATA_BLOCK

DATA_BLOCK "S1.CABINET033.WARNING2"   // DB2335
// stored: AutoNumber true, DBAccessibleFromOPCUA true, DBAccessibleFromWebserver true, InstanceOfName BoolToUDInt_Inverted_Filtered, InstanceOfType FB
"BoolToUDInt_Inverted_Filtered "
BEGIN
END_DATA_BLOCK

DATA_BLOCK "S1.CABINET034.ALARM1"   // DB2336
// stored: AutoNumber true, DBAccessibleFromOPCUA true, DBAccessibleFromWebserver true, InstanceOfName BoolToUDInt_Inverted_Filtered, InstanceOfType FB
"BoolToUDInt_Inverted_Filtered "
BEGIN
END_DATA_BLOCK

DATA_BLOCK "S1.CABINET034.ALARM2"   // DB2337
// stored: AutoNumber true, DBAccessibleFromOPCUA true, DBAccessibleFromWebserver true, InstanceOfName BoolToUDInt_Inverted_Filtered, InstanceOfType FB
"BoolToUDInt_Inverted_Filtered "
BEGIN
END_DATA_BLOCK

DATA_BLOCK "S1.CABINET034.WARNING1"   // DB2338
// stored: AutoNumber true, DBAccessibleFromOPCUA true, DBAccessibleFromWebserver true, InstanceOfName BoolToUDInt_Inverted_Filtered, InstanceOfType FB
"BoolToUDInt_Inverted_Filtered "
BEGIN
END_DATA_BLOCK

DATA_BLOCK "S1.CABINET034.WARNING2"   // DB2339
// stored: AutoNumber true, DBAccessibleFromOPCUA true, DBAccessibleFromWebserver true, InstanceOfName BoolToUDInt_Inverted_Filtered, InstanceOfType FB
"BoolToUDInt_Inverted_Filtered "
BEGIN
END_DATA_BLOCK

DATA_BLOCK "S1.CABINET035.ALARM1"   // DB2340
// stored: AutoNumber true, DBAccessibleFromOPCUA true, DBAccessibleFromWebserver true, InstanceOfName BoolToUDInt_Inverted_Filtered, InstanceOfType FB
"BoolToUDInt_Inverted_Filtered "
BEGIN
END_DATA_BLOCK

DATA_BLOCK "S1.CABINET035.ALARM2"   // DB2341
// stored: AutoNumber true, DBAccessibleFromOPCUA true, DBAccessibleFromWebserver true, InstanceOfName BoolToUDInt_Inverted_Filtered, InstanceOfType FB
"BoolToUDInt_Inverted_Filtered "
BEGIN
END_DATA_BLOCK

DATA_BLOCK "S1.CABINET035.WARNING1"   // DB2342
// stored: AutoNumber true, DBAccessibleFromOPCUA true, DBAccessibleFromWebserver true, InstanceOfName BoolToUDInt_Inverted_Filtered, InstanceOfType FB
"BoolToUDInt_Inverted_Filtered "
BEGIN
END_DATA_BLOCK

DATA_BLOCK "S1.CABINET035.WARNING2"   // DB2343
// stored: AutoNumber true, DBAccessibleFromOPCUA true, DBAccessibleFromWebserver true, InstanceOfName BoolToUDInt_Inverted_Filtered, InstanceOfType FB
"BoolToUDInt_Inverted_Filtered "
BEGIN
END_DATA_BLOCK

DATA_BLOCK "S1.CABINET036.ALARM1"   // DB2344
// stored: AutoNumber true, DBAccessibleFromOPCUA true, DBAccessibleFromWebserver true, InstanceOfName BoolToUDInt_Inverted_Filtered, InstanceOfType FB
"BoolToUDInt_Inverted_Filtered "
BEGIN
END_DATA_BLOCK

DATA_BLOCK "S1.CABINET036.ALARM2"   // DB2345
// stored: AutoNumber true, DBAccessibleFromOPCUA true, DBAccessibleFromWebserver true, InstanceOfName BoolToUDInt_Inverted_Filtered, InstanceOfType FB
"BoolToUDInt_Inverted_Filtered "
BEGIN
END_DATA_BLOCK

DATA_BLOCK "S1.CABINET036.WARNING1"   // DB2346
// stored: AutoNumber true, DBAccessibleFromOPCUA true, DBAccessibleFromWebserver true, InstanceOfName BoolToUDInt_Inverted_Filtered, InstanceOfType FB
"BoolToUDInt_Inverted_Filtered "
BEGIN
END_DATA_BLOCK

DATA_BLOCK "S1.CABINET036.WARNING2"   // DB2347
// stored: AutoNumber true, DBAccessibleFromOPCUA true, DBAccessibleFromWebserver true, InstanceOfName BoolToUDInt_Inverted_Filtered, InstanceOfType FB
"BoolToUDInt_Inverted_Filtered "
BEGIN
END_DATA_BLOCK

DATA_BLOCK "S1.CABINET037.ALARM1"   // DB2348
// stored: AutoNumber true, DBAccessibleFromOPCUA true, DBAccessibleFromWebserver true, InstanceOfName BoolToUDInt_Inverted_Filtered, InstanceOfType FB
"BoolToUDInt_Inverted_Filtered "
BEGIN
END_DATA_BLOCK

DATA_BLOCK "S1.CABINET037.ALARM2"   // DB2349
// stored: AutoNumber true, DBAccessibleFromOPCUA true, DBAccessibleFromWebserver true, InstanceOfName BoolToUDInt_Inverted_Filtered, InstanceOfType FB
"BoolToUDInt_Inverted_Filtered "
BEGIN
END_DATA_BLOCK

DATA_BLOCK "S1.CABINET037.WARNING1"   // DB2350
// stored: AutoNumber true, DBAccessibleFromOPCUA true, DBAccessibleFromWebserver true, InstanceOfName BoolToUDInt_Inverted_Filtered, InstanceOfType FB
"BoolToUDInt_Inverted_Filtered "
BEGIN
END_DATA_BLOCK

DATA_BLOCK "S1.CABINET037.WARNING2"   // DB2351
// stored: AutoNumber true, DBAccessibleFromOPCUA true, DBAccessibleFromWebserver true, InstanceOfName BoolToUDInt_Inverted_Filtered, InstanceOfType FB
"BoolToUDInt_Inverted_Filtered "
BEGIN
END_DATA_BLOCK

DATA_BLOCK "S1.CABINET038.ALARM1"   // DB2352
// stored: AutoNumber true, DBAccessibleFromOPCUA true, DBAccessibleFromWebserver true, InstanceOfName BoolToUDInt_Inverted_Filtered, InstanceOfType FB
"BoolToUDInt_Inverted_Filtered "
BEGIN
END_DATA_BLOCK

DATA_BLOCK "S1.CABINET038.ALARM2"   // DB2353
// stored: AutoNumber true, DBAccessibleFromOPCUA true, DBAccessibleFromWebserver true, InstanceOfName BoolToUDInt_Inverted_Filtered, InstanceOfType FB
"BoolToUDInt_Inverted_Filtered "
BEGIN
END_DATA_BLOCK

DATA_BLOCK "S1.CABINET038.WARNING1"   // DB2354
// stored: AutoNumber true, DBAccessibleFromOPCUA true, DBAccessibleFromWebserver true, InstanceOfName BoolToUDInt_Inverted_Filtered, InstanceOfType FB
"BoolToUDInt_Inverted_Filtered "
BEGIN
END_DATA_BLOCK

DATA_BLOCK "S1.CABINET038.WARNING2"   // DB2355
// stored: AutoNumber true, DBAccessibleFromOPCUA true, DBAccessibleFromWebserver true, InstanceOfName BoolToUDInt_Inverted_Filtered, InstanceOfType FB
"BoolToUDInt_Inverted_Filtered "
BEGIN
END_DATA_BLOCK

DATA_BLOCK "S1.CABINET039.ALARM1"   // DB2356
// stored: AutoNumber true, DBAccessibleFromOPCUA true, DBAccessibleFromWebserver true, InstanceOfName BoolToUDInt_Inverted_Filtered, InstanceOfType FB
"BoolToUDInt_Inverted_Filtered "
BEGIN
END_DATA_BLOCK

DATA_BLOCK "S1.CABINET039.ALARM2"   // DB2357
// stored: AutoNumber true, DBAccessibleFromOPCUA true, DBAccessibleFromWebserver true, InstanceOfName BoolToUDInt_Inverted_Filtered, InstanceOfType FB
"BoolToUDInt_Inverted_Filtered "
BEGIN
END_DATA_BLOCK

DATA_BLOCK "S1.CABINET039.WARNING1"   // DB2358
// stored: AutoNumber true, DBAccessibleFromOPCUA true, DBAccessibleFromWebserver true, InstanceOfName BoolToUDInt_Inverted_Filtered, InstanceOfType FB
"BoolToUDInt_Inverted_Filtered "
BEGIN
END_DATA_BLOCK

DATA_BLOCK "S1.CABINET039.WARNING2"   // DB2359
// stored: AutoNumber true, DBAccessibleFromOPCUA true, DBAccessibleFromWebserver true, InstanceOfName BoolToUDInt_Inverted_Filtered, InstanceOfType FB
"BoolToUDInt_Inverted_Filtered "
BEGIN
END_DATA_BLOCK

DATA_BLOCK "S1.CABINET040.ALARM1"   // DB2360
// stored: AutoNumber true, DBAccessibleFromOPCUA true, DBAccessibleFromWebserver true, InstanceOfName BoolToUDInt_Inverted_Filtered, InstanceOfType FB
"BoolToUDInt_Inverted_Filtered "
BEGIN
END_DATA_BLOCK

DATA_BLOCK "S1.CABINET040.ALARM2"   // DB2361
// stored: AutoNumber true, DBAccessibleFromOPCUA true, DBAccessibleFromWebserver true, InstanceOfName BoolToUDInt_Inverted_Filtered, InstanceOfType FB
"BoolToUDInt_Inverted_Filtered "
BEGIN
END_DATA_BLOCK

DATA_BLOCK "S1.CABINET040.WARNING1"   // DB2362
// stored: AutoNumber true, DBAccessibleFromOPCUA true, DBAccessibleFromWebserver true, InstanceOfName BoolToUDInt_Inverted_Filtered, InstanceOfType FB
"BoolToUDInt_Inverted_Filtered "
BEGIN
END_DATA_BLOCK

DATA_BLOCK "S1.CABINET040.WARNING2"   // DB2363
// stored: AutoNumber true, DBAccessibleFromOPCUA true, DBAccessibleFromWebserver true, InstanceOfName BoolToUDInt_Inverted_Filtered, InstanceOfType FB
"BoolToUDInt_Inverted_Filtered "
BEGIN
END_DATA_BLOCK

DATA_BLOCK "S1.CABINET041.ALARM1"   // DB2364
// stored: AutoNumber true, DBAccessibleFromOPCUA true, DBAccessibleFromWebserver true, InstanceOfName BoolToUDInt_Inverted_Filtered, InstanceOfType FB
"BoolToUDInt_Inverted_Filtered "
BEGIN
END_DATA_BLOCK

DATA_BLOCK "S1.CABINET041.ALARM2"   // DB2365
// stored: AutoNumber true, DBAccessibleFromOPCUA true, DBAccessibleFromWebserver true, InstanceOfName BoolToUDInt_Inverted_Filtered, InstanceOfType FB
"BoolToUDInt_Inverted_Filtered "
BEGIN
END_DATA_BLOCK

DATA_BLOCK "S1.CABINET041.WARNING1"   // DB2366
// stored: AutoNumber true, DBAccessibleFromOPCUA true, DBAccessibleFromWebserver true, InstanceOfName BoolToUDInt_Inverted_Filtered, InstanceOfType FB
"BoolToUDInt_Inverted_Filtered "
BEGIN
END_DATA_BLOCK

DATA_BLOCK "S1.CABINET041.WARNING2"   // DB2367
// stored: AutoNumber true, DBAccessibleFromOPCUA true, DBAccessibleFromWebserver true, InstanceOfName BoolToUDInt_Inverted_Filtered, InstanceOfType FB
"BoolToUDInt_Inverted_Filtered "
BEGIN
END_DATA_BLOCK

DATA_BLOCK "S1.CABINET042.ALARM1"   // DB2368
// stored: AutoNumber true, DBAccessibleFromOPCUA true, DBAccessibleFromWebserver true, InstanceOfName BoolToUDInt_Inverted_Filtered, InstanceOfType FB
"BoolToUDInt_Inverted_Filtered "
BEGIN
END_DATA_BLOCK

DATA_BLOCK "S1.CABINET042.ALARM2"   // DB2369
// stored: AutoNumber true, DBAccessibleFromOPCUA true, DBAccessibleFromWebserver true, InstanceOfName BoolToUDInt_Inverted_Filtered, InstanceOfType FB
"BoolToUDInt_Inverted_Filtered "
BEGIN
END_DATA_BLOCK

DATA_BLOCK "S1.CABINET042.WARNING1"   // DB2370
// stored: AutoNumber true, DBAccessibleFromOPCUA true, DBAccessibleFromWebserver true, InstanceOfName BoolToUDInt_Inverted_Filtered, InstanceOfType FB
"BoolToUDInt_Inverted_Filtered "
BEGIN
END_DATA_BLOCK

DATA_BLOCK "S1.CABINET042.WARNING2"   // DB2371
// stored: AutoNumber true, DBAccessibleFromOPCUA true, DBAccessibleFromWebserver true, InstanceOfName BoolToUDInt_Inverted_Filtered, InstanceOfType FB
"BoolToUDInt_Inverted_Filtered "
BEGIN
END_DATA_BLOCK

DATA_BLOCK "S1.CABINET043.ALARM1"   // DB2372
// stored: AutoNumber true, DBAccessibleFromOPCUA true, DBAccessibleFromWebserver true, InstanceOfName BoolToUDInt_Inverted_Filtered, InstanceOfType FB
"BoolToUDInt_Inverted_Filtered "
BEGIN
END_DATA_BLOCK

DATA_BLOCK "S1.CABINET043.ALARM2"   // DB2373
// stored: AutoNumber true, DBAccessibleFromOPCUA true, DBAccessibleFromWebserver true, InstanceOfName BoolToUDInt_Inverted_Filtered, InstanceOfType FB
"BoolToUDInt_Inverted_Filtered "
BEGIN
END_DATA_BLOCK

DATA_BLOCK "S1.CABINET043.WARNING1"   // DB2374
// stored: AutoNumber true, DBAccessibleFromOPCUA true, DBAccessibleFromWebserver true, InstanceOfName BoolToUDInt_Inverted_Filtered, InstanceOfType FB
"BoolToUDInt_Inverted_Filtered "
BEGIN
END_DATA_BLOCK

DATA_BLOCK "S1.CABINET043.WARNING2"   // DB2375
// stored: AutoNumber true, DBAccessibleFromOPCUA true, DBAccessibleFromWebserver true, InstanceOfName BoolToUDInt_Inverted_Filtered, InstanceOfType FB
"BoolToUDInt_Inverted_Filtered "
BEGIN
END_DATA_BLOCK

DATA_BLOCK "S1.CABINET044.ALARM1"   // DB2376
// stored: AutoNumber true, DBAccessibleFromOPCUA true, DBAccessibleFromWebserver true, InstanceOfName BoolToUDInt_Inverted_Filtered, InstanceOfType FB
"BoolToUDInt_Inverted_Filtered "
BEGIN
END_DATA_BLOCK

DATA_BLOCK "S1.CABINET044.ALARM2"   // DB2377
// stored: AutoNumber true, DBAccessibleFromOPCUA true, DBAccessibleFromWebserver true, InstanceOfName BoolToUDInt_Inverted_Filtered, InstanceOfType FB
"BoolToUDInt_Inverted_Filtered "
BEGIN
END_DATA_BLOCK

DATA_BLOCK "S1.CABINET044.WARNING1"   // DB2378
// stored: AutoNumber true, DBAccessibleFromOPCUA true, DBAccessibleFromWebserver true, InstanceOfName BoolToUDInt_Inverted_Filtered, InstanceOfType FB
"BoolToUDInt_Inverted_Filtered "
BEGIN
END_DATA_BLOCK

DATA_BLOCK "S1.CABINET044.WARNING2"   // DB2379
// stored: AutoNumber true, DBAccessibleFromOPCUA true, DBAccessibleFromWebserver true, InstanceOfName BoolToUDInt_Inverted_Filtered, InstanceOfType FB
"BoolToUDInt_Inverted_Filtered "
BEGIN
END_DATA_BLOCK

DATA_BLOCK "S1.CABINET045.ALARM1"   // DB2380
// stored: AutoNumber true, DBAccessibleFromOPCUA true, DBAccessibleFromWebserver true, InstanceOfName BoolToUDInt_Inverted_Filtered, InstanceOfType FB
"BoolToUDInt_Inverted_Filtered "
BEGIN
END_DATA_BLOCK

DATA_BLOCK "S1.CABINET045.ALARM2"   // DB2381
// stored: AutoNumber true, DBAccessibleFromOPCUA true, DBAccessibleFromWebserver true, InstanceOfName BoolToUDInt_Inverted_Filtered, InstanceOfType FB
"BoolToUDInt_Inverted_Filtered "
BEGIN
END_DATA_BLOCK

DATA_BLOCK "S1.CABINET045.WARNING1"   // DB2382
// stored: AutoNumber true, DBAccessibleFromOPCUA true, DBAccessibleFromWebserver true, InstanceOfName BoolToUDInt_Inverted_Filtered, InstanceOfType FB
"BoolToUDInt_Inverted_Filtered "
BEGIN
END_DATA_BLOCK

DATA_BLOCK "S1.CABINET045.WARNING2"   // DB2383
// stored: AutoNumber true, DBAccessibleFromOPCUA true, DBAccessibleFromWebserver true, InstanceOfName BoolToUDInt_Inverted_Filtered, InstanceOfType FB
"BoolToUDInt_Inverted_Filtered "
BEGIN
END_DATA_BLOCK

DATA_BLOCK "S1.CABINET046.ALARM1"   // DB2384
// stored: AutoNumber true, DBAccessibleFromOPCUA true, DBAccessibleFromWebserver true, InstanceOfName BoolToUDInt_Inverted_Filtered, InstanceOfType FB
"BoolToUDInt_Inverted_Filtered "
BEGIN
END_DATA_BLOCK

DATA_BLOCK "S1.CABINET046.ALARM2"   // DB2385
// stored: AutoNumber true, DBAccessibleFromOPCUA true, DBAccessibleFromWebserver true, InstanceOfName BoolToUDInt_Inverted_Filtered, InstanceOfType FB
"BoolToUDInt_Inverted_Filtered "
BEGIN
END_DATA_BLOCK

DATA_BLOCK "S1.CABINET046.WARNING1"   // DB2386
// stored: AutoNumber true, DBAccessibleFromOPCUA true, DBAccessibleFromWebserver true, InstanceOfName BoolToUDInt_Inverted_Filtered, InstanceOfType FB
"BoolToUDInt_Inverted_Filtered "
BEGIN
END_DATA_BLOCK

DATA_BLOCK "S1.CABINET046.WARNING2"   // DB2387
// stored: AutoNumber true, DBAccessibleFromOPCUA true, DBAccessibleFromWebserver true, InstanceOfName BoolToUDInt_Inverted_Filtered, InstanceOfType FB
"BoolToUDInt_Inverted_Filtered "
BEGIN
END_DATA_BLOCK

DATA_BLOCK "S1.CABINET047.ALARM1"   // DB2388
// stored: AutoNumber true, DBAccessibleFromOPCUA true, DBAccessibleFromWebserver true, InstanceOfName BoolToUDInt_Inverted_Filtered, InstanceOfType FB
"BoolToUDInt_Inverted_Filtered "
BEGIN
END_DATA_BLOCK

DATA_BLOCK "S1.CABINET047.ALARM2"   // DB2389
// stored: AutoNumber true, DBAccessibleFromOPCUA true, DBAccessibleFromWebserver true, InstanceOfName BoolToUDInt_Inverted_Filtered, InstanceOfType FB
"BoolToUDInt_Inverted_Filtered "
BEGIN
END_DATA_BLOCK

DATA_BLOCK "S1.CABINET047.WARNING1"   // DB2390
// stored: AutoNumber true, DBAccessibleFromOPCUA true, DBAccessibleFromWebserver true, InstanceOfName BoolToUDInt_Inverted_Filtered, InstanceOfType FB
"BoolToUDInt_Inverted_Filtered "
BEGIN
END_DATA_BLOCK

DATA_BLOCK "S1.CABINET047.WARNING2"   // DB2391
// stored: AutoNumber true, DBAccessibleFromOPCUA true, DBAccessibleFromWebserver true, InstanceOfName BoolToUDInt_Inverted_Filtered, InstanceOfType FB
"BoolToUDInt_Inverted_Filtered "
BEGIN
END_DATA_BLOCK

DATA_BLOCK "S1.CABINET048.ALARM1"   // DB2392
// stored: AutoNumber true, DBAccessibleFromOPCUA true, DBAccessibleFromWebserver true, InstanceOfName BoolToUDInt_Inverted_Filtered, InstanceOfType FB
"BoolToUDInt_Inverted_Filtered "
BEGIN
END_DATA_BLOCK

DATA_BLOCK "S1.CABINET048.ALARM2"   // DB2393
// stored: AutoNumber true, DBAccessibleFromOPCUA true, DBAccessibleFromWebserver true, InstanceOfName BoolToUDInt_Inverted_Filtered, InstanceOfType FB
"BoolToUDInt_Inverted_Filtered "
BEGIN
END_DATA_BLOCK

DATA_BLOCK "S1.CABINET048.WARNING1"   // DB2394
// stored: AutoNumber true, DBAccessibleFromOPCUA true, DBAccessibleFromWebserver true, InstanceOfName BoolToUDInt_Inverted_Filtered, InstanceOfType FB
"BoolToUDInt_Inverted_Filtered "
BEGIN
END_DATA_BLOCK

DATA_BLOCK "S1.CABINET048.WARNING2"   // DB2395
// stored: AutoNumber true, DBAccessibleFromOPCUA true, DBAccessibleFromWebserver true, InstanceOfName BoolToUDInt_Inverted_Filtered, InstanceOfType FB
"BoolToUDInt_Inverted_Filtered "
BEGIN
END_DATA_BLOCK

DATA_BLOCK "S1.CABINET049.ALARM1"   // DB2396
// stored: AutoNumber true, DBAccessibleFromOPCUA true, DBAccessibleFromWebserver true, InstanceOfName BoolToUDInt_Inverted_Filtered, InstanceOfType FB
"BoolToUDInt_Inverted_Filtered "
BEGIN
END_DATA_BLOCK

DATA_BLOCK "S1.CABINET049.ALARM2"   // DB2397
// stored: AutoNumber true, DBAccessibleFromOPCUA true, DBAccessibleFromWebserver true, InstanceOfName BoolToUDInt_Inverted_Filtered, InstanceOfType FB
"BoolToUDInt_Inverted_Filtered "
BEGIN
END_DATA_BLOCK

DATA_BLOCK "S1.CABINET049.WARNING1"   // DB2398
// stored: AutoNumber true, DBAccessibleFromOPCUA true, DBAccessibleFromWebserver true, InstanceOfName BoolToUDInt_Inverted_Filtered, InstanceOfType FB
"BoolToUDInt_Inverted_Filtered "
BEGIN
END_DATA_BLOCK

DATA_BLOCK "S1.CABINET049.WARNING2"   // DB2399
// stored: AutoNumber true, DBAccessibleFromOPCUA true, DBAccessibleFromWebserver true, InstanceOfName BoolToUDInt_Inverted_Filtered, InstanceOfType FB
"BoolToUDInt_Inverted_Filtered "
BEGIN
END_DATA_BLOCK

DATA_BLOCK "S1.CABINET050.ALARM1"   // DB2400
// stored: AutoNumber true, DBAccessibleFromOPCUA true, DBAccessibleFromWebserver true, InstanceOfName BoolToUDInt_Inverted_Filtered, InstanceOfType FB
"BoolToUDInt_Inverted_Filtered "
BEGIN
END_DATA_BLOCK

DATA_BLOCK "S1.CABINET050.ALARM2"   // DB2401
// stored: AutoNumber true, DBAccessibleFromOPCUA true, DBAccessibleFromWebserver true, InstanceOfName BoolToUDInt_Inverted_Filtered, InstanceOfType FB
"BoolToUDInt_Inverted_Filtered "
BEGIN
END_DATA_BLOCK

DATA_BLOCK "S1.CABINET050.WARNING1"   // DB2402
// stored: AutoNumber true, DBAccessibleFromOPCUA true, DBAccessibleFromWebserver true, InstanceOfName BoolToUDInt_Inverted_Filtered, InstanceOfType FB
"BoolToUDInt_Inverted_Filtered "
BEGIN
END_DATA_BLOCK

DATA_BLOCK "S1.CABINET050.WARNING2"   // DB2403
// stored: AutoNumber true, DBAccessibleFromOPCUA true, DBAccessibleFromWebserver true, InstanceOfName BoolToUDInt_Inverted_Filtered, InstanceOfType FB
"BoolToUDInt_Inverted_Filtered "
BEGIN
END_DATA_BLOCK

DATA_BLOCK "S1.CABINET051.ALARM1"   // DB2404
// stored: AutoNumber true, DBAccessibleFromOPCUA true, DBAccessibleFromWebserver true, InstanceOfName BoolToUDInt_Inverted_Filtered, InstanceOfType FB
"BoolToUDInt_Inverted_Filtered "
BEGIN
END_DATA_BLOCK

DATA_BLOCK "S1.CABINET051.ALARM2"   // DB2405
// stored: AutoNumber true, DBAccessibleFromOPCUA true, DBAccessibleFromWebserver true, InstanceOfName BoolToUDInt_Inverted_Filtered, InstanceOfType FB
"BoolToUDInt_Inverted_Filtered "
BEGIN
END_DATA_BLOCK

DATA_BLOCK "S1.CABINET051.WARNING1"   // DB2406
// stored: AutoNumber true, DBAccessibleFromOPCUA true, DBAccessibleFromWebserver true, InstanceOfName BoolToUDInt_Inverted_Filtered, InstanceOfType FB
"BoolToUDInt_Inverted_Filtered "
BEGIN
END_DATA_BLOCK

DATA_BLOCK "S1.CABINET051.WARNING2"   // DB2407
// stored: AutoNumber true, DBAccessibleFromOPCUA true, DBAccessibleFromWebserver true, InstanceOfName BoolToUDInt_Inverted_Filtered, InstanceOfType FB
"BoolToUDInt_Inverted_Filtered "
BEGIN
END_DATA_BLOCK

DATA_BLOCK "S1.CABINET052.ALARM1"   // DB2408
// stored: AutoNumber true, DBAccessibleFromOPCUA true, DBAccessibleFromWebserver true, InstanceOfName BoolToUDInt_Inverted_Filtered, InstanceOfType FB
"BoolToUDInt_Inverted_Filtered "
BEGIN
END_DATA_BLOCK

DATA_BLOCK "S1.CABINET052.ALARM2"   // DB2409
// stored: AutoNumber true, DBAccessibleFromOPCUA true, DBAccessibleFromWebserver true, InstanceOfName BoolToUDInt_Inverted_Filtered, InstanceOfType FB
"BoolToUDInt_Inverted_Filtered "
BEGIN
END_DATA_BLOCK

DATA_BLOCK "S1.CABINET052.WARNING1"   // DB2410
// stored: AutoNumber true, DBAccessibleFromOPCUA true, DBAccessibleFromWebserver true, InstanceOfName BoolToUDInt_Inverted_Filtered, InstanceOfType FB
"BoolToUDInt_Inverted_Filtered "
BEGIN
END_DATA_BLOCK

DATA_BLOCK "S1.CABINET052.WARNING2"   // DB2411
// stored: AutoNumber true, DBAccessibleFromOPCUA true, DBAccessibleFromWebserver true, InstanceOfName BoolToUDInt_Inverted_Filtered, InstanceOfType FB
"BoolToUDInt_Inverted_Filtered "
BEGIN
END_DATA_BLOCK

DATA_BLOCK "S1.CABINET053.ALARM1"   // DB2412
// stored: AutoNumber true, DBAccessibleFromOPCUA true, DBAccessibleFromWebserver true, InstanceOfName BoolToUDInt_Inverted_Filtered, InstanceOfType FB
"BoolToUDInt_Inverted_Filtered "
BEGIN
END_DATA_BLOCK

DATA_BLOCK "S1.CABINET053.ALARM2"   // DB2413
// stored: AutoNumber true, DBAccessibleFromOPCUA true, DBAccessibleFromWebserver true, InstanceOfName BoolToUDInt_Inverted_Filtered, InstanceOfType FB
"BoolToUDInt_Inverted_Filtered "
BEGIN
END_DATA_BLOCK

DATA_BLOCK "S1.CABINET053.WARNING1"   // DB2414
// stored: AutoNumber true, DBAccessibleFromOPCUA true, DBAccessibleFromWebserver true, InstanceOfName BoolToUDInt_Inverted_Filtered, InstanceOfType FB
"BoolToUDInt_Inverted_Filtered "
BEGIN
END_DATA_BLOCK

DATA_BLOCK "S1.CABINET053.WARNING2"   // DB2415
// stored: AutoNumber true, DBAccessibleFromOPCUA true, DBAccessibleFromWebserver true, InstanceOfName BoolToUDInt_Inverted_Filtered, InstanceOfType FB
"BoolToUDInt_Inverted_Filtered "
BEGIN
END_DATA_BLOCK

DATA_BLOCK "S1.CABINET054.ALARM1"   // DB2416
// stored: AutoNumber true, DBAccessibleFromOPCUA true, DBAccessibleFromWebserver true, InstanceOfName BoolToUDInt_Inverted_Filtered, InstanceOfType FB
"BoolToUDInt_Inverted_Filtered "
BEGIN
END_DATA_BLOCK

DATA_BLOCK "S1.CABINET054.ALARM2"   // DB2417
// stored: AutoNumber true, DBAccessibleFromOPCUA true, DBAccessibleFromWebserver true, InstanceOfName BoolToUDInt_Inverted_Filtered, InstanceOfType FB
"BoolToUDInt_Inverted_Filtered "
BEGIN
END_DATA_BLOCK

DATA_BLOCK "S1.CABINET054.WARNING1"   // DB2418
// stored: AutoNumber true, DBAccessibleFromOPCUA true, DBAccessibleFromWebserver true, InstanceOfName BoolToUDInt_Inverted_Filtered, InstanceOfType FB
"BoolToUDInt_Inverted_Filtered "
BEGIN
END_DATA_BLOCK

DATA_BLOCK "S1.CABINET054.WARNING2"   // DB2419
// stored: AutoNumber true, DBAccessibleFromOPCUA true, DBAccessibleFromWebserver true, InstanceOfName BoolToUDInt_Inverted_Filtered, InstanceOfType FB
"BoolToUDInt_Inverted_Filtered "
BEGIN
END_DATA_BLOCK

DATA_BLOCK "S1.CABINET055.ALARM1"   // DB2420
// stored: AutoNumber true, DBAccessibleFromOPCUA true, DBAccessibleFromWebserver true, InstanceOfName BoolToUDInt_Inverted_Filtered, InstanceOfType FB
"BoolToUDInt_Inverted_Filtered "
BEGIN
END_DATA_BLOCK

DATA_BLOCK "S1.CABINET055.ALARM2"   // DB2421
// stored: AutoNumber true, DBAccessibleFromOPCUA true, DBAccessibleFromWebserver true, InstanceOfName BoolToUDInt_Inverted_Filtered, InstanceOfType FB
"BoolToUDInt_Inverted_Filtered "
BEGIN
END_DATA_BLOCK

DATA_BLOCK "S1.CABINET055.WARNING1"   // DB2422
// stored: AutoNumber true, DBAccessibleFromOPCUA true, DBAccessibleFromWebserver true, InstanceOfName BoolToUDInt_Inverted_Filtered, InstanceOfType FB
"BoolToUDInt_Inverted_Filtered "
BEGIN
END_DATA_BLOCK

DATA_BLOCK "S1.CABINET055.WARNING2"   // DB2423
// stored: AutoNumber true, DBAccessibleFromOPCUA true, DBAccessibleFromWebserver true, InstanceOfName BoolToUDInt_Inverted_Filtered, InstanceOfType FB
"BoolToUDInt_Inverted_Filtered "
BEGIN
END_DATA_BLOCK

DATA_BLOCK "S1.CABINET056.ALARM1"   // DB2424
// stored: AutoNumber true, DBAccessibleFromOPCUA true, DBAccessibleFromWebserver true, InstanceOfName BoolToUDInt_Inverted_Filtered, InstanceOfType FB
"BoolToUDInt_Inverted_Filtered "
BEGIN
END_DATA_BLOCK

DATA_BLOCK "S1.CABINET056.ALARM2"   // DB2425
// stored: AutoNumber true, DBAccessibleFromOPCUA true, DBAccessibleFromWebserver true, InstanceOfName BoolToUDInt_Inverted_Filtered, InstanceOfType FB
"BoolToUDInt_Inverted_Filtered "
BEGIN
END_DATA_BLOCK

DATA_BLOCK "S1.CABINET056.WARNING1"   // DB2426
// stored: AutoNumber true, DBAccessibleFromOPCUA true, DBAccessibleFromWebserver true, InstanceOfName BoolToUDInt_Inverted_Filtered, InstanceOfType FB
"BoolToUDInt_Inverted_Filtered "
BEGIN
END_DATA_BLOCK

DATA_BLOCK "S1.CABINET056.WARNING2"   // DB2427
// stored: AutoNumber true, DBAccessibleFromOPCUA true, DBAccessibleFromWebserver true, InstanceOfName BoolToUDInt_Inverted_Filtered, InstanceOfType FB
"BoolToUDInt_Inverted_Filtered "
BEGIN
END_DATA_BLOCK

DATA_BLOCK "S1.CABINET057.ALARM1"   // DB2428
// stored: AutoNumber true, DBAccessibleFromOPCUA true, DBAccessibleFromWebserver true, InstanceOfName BoolToUDInt_Inverted_Filtered, InstanceOfType FB
"BoolToUDInt_Inverted_Filtered "
BEGIN
END_DATA_BLOCK

DATA_BLOCK "S1.CABINET057.ALARM2"   // DB2429
// stored: AutoNumber true, DBAccessibleFromOPCUA true, DBAccessibleFromWebserver true, InstanceOfName BoolToUDInt_Inverted_Filtered, InstanceOfType FB
"BoolToUDInt_Inverted_Filtered "
BEGIN
END_DATA_BLOCK

DATA_BLOCK "S1.CABINET057.WARNING1"   // DB2430
// stored: AutoNumber true, DBAccessibleFromOPCUA true, DBAccessibleFromWebserver true, InstanceOfName BoolToUDInt_Inverted_Filtered, InstanceOfType FB
"BoolToUDInt_Inverted_Filtered "
BEGIN
END_DATA_BLOCK

DATA_BLOCK "S1.CABINET057.WARNING2"   // DB2431
// stored: AutoNumber true, DBAccessibleFromOPCUA true, DBAccessibleFromWebserver true, InstanceOfName BoolToUDInt_Inverted_Filtered, InstanceOfType FB
"BoolToUDInt_Inverted_Filtered "
BEGIN
END_DATA_BLOCK

DATA_BLOCK "S1.CABINET058.ALARM1"   // DB2432
// stored: AutoNumber true, DBAccessibleFromOPCUA true, DBAccessibleFromWebserver true, InstanceOfName BoolToUDInt_Inverted_Filtered, InstanceOfType FB
"BoolToUDInt_Inverted_Filtered "
BEGIN
END_DATA_BLOCK

DATA_BLOCK "S1.CABINET058.ALARM2"   // DB2433
// stored: AutoNumber true, DBAccessibleFromOPCUA true, DBAccessibleFromWebserver true, InstanceOfName BoolToUDInt_Inverted_Filtered, InstanceOfType FB
"BoolToUDInt_Inverted_Filtered "
BEGIN
END_DATA_BLOCK

DATA_BLOCK "S1.CABINET058.WARNING1"   // DB2434
// stored: AutoNumber true, DBAccessibleFromOPCUA true, DBAccessibleFromWebserver true, InstanceOfName BoolToUDInt_Inverted_Filtered, InstanceOfType FB
"BoolToUDInt_Inverted_Filtered "
BEGIN
END_DATA_BLOCK

DATA_BLOCK "S1.CABINET058.WARNING2"   // DB2435
// stored: AutoNumber true, DBAccessibleFromOPCUA true, DBAccessibleFromWebserver true, InstanceOfName BoolToUDInt_Inverted_Filtered, InstanceOfType FB
"BoolToUDInt_Inverted_Filtered "
BEGIN
END_DATA_BLOCK

DATA_BLOCK "S1.CABINET059.ALARM1"   // DB2436
// stored: AutoNumber true, DBAccessibleFromOPCUA true, DBAccessibleFromWebserver true, InstanceOfName BoolToUDInt_Inverted_Filtered, InstanceOfType FB
"BoolToUDInt_Inverted_Filtered "
BEGIN
END_DATA_BLOCK

DATA_BLOCK "S1.CABINET059.ALARM2"   // DB2437
// stored: AutoNumber true, DBAccessibleFromOPCUA true, DBAccessibleFromWebserver true, InstanceOfName BoolToUDInt_Inverted_Filtered, InstanceOfType FB
"BoolToUDInt_Inverted_Filtered "
BEGIN
END_DATA_BLOCK

DATA_BLOCK "S1.CABINET059.WARNING1"   // DB2438
// stored: AutoNumber true, DBAccessibleFromOPCUA true, DBAccessibleFromWebserver true, InstanceOfName BoolToUDInt_Inverted_Filtered, InstanceOfType FB
"BoolToUDInt_Inverted_Filtered "
BEGIN
END_DATA_BLOCK

DATA_BLOCK "S1.CABINET059.WARNING2"   // DB2439
// stored: AutoNumber true, DBAccessibleFromOPCUA true, DBAccessibleFromWebserver true, InstanceOfName BoolToUDInt_Inverted_Filtered, InstanceOfType FB
"BoolToUDInt_Inverted_Filtered "
BEGIN
END_DATA_BLOCK

DATA_BLOCK "S1.CABINET060.ALARM1"   // DB2440
// stored: AutoNumber true, DBAccessibleFromOPCUA true, DBAccessibleFromWebserver true, InstanceOfName BoolToUDInt_Inverted_Filtered, InstanceOfType FB
"BoolToUDInt_Inverted_Filtered "
BEGIN
END_DATA_BLOCK

DATA_BLOCK "S1.CABINET060.ALARM2"   // DB2441
// stored: AutoNumber true, DBAccessibleFromOPCUA true, DBAccessibleFromWebserver true, InstanceOfName BoolToUDInt_Inverted_Filtered, InstanceOfType FB
"BoolToUDInt_Inverted_Filtered "
BEGIN
END_DATA_BLOCK

DATA_BLOCK "S1.CABINET060.WARNING1"   // DB2442
// stored: AutoNumber true, DBAccessibleFromOPCUA true, DBAccessibleFromWebserver true, InstanceOfName BoolToUDInt_Inverted_Filtered, InstanceOfType FB
"BoolToUDInt_Inverted_Filtered "
BEGIN
END_DATA_BLOCK

DATA_BLOCK "S1.CABINET060.WARNING2"   // DB2443
// stored: AutoNumber true, DBAccessibleFromOPCUA true, DBAccessibleFromWebserver true, InstanceOfName BoolToUDInt_Inverted_Filtered, InstanceOfType FB
"BoolToUDInt_Inverted_Filtered "
BEGIN
END_DATA_BLOCK

DATA_BLOCK "S1.CABINET061.ALARM1"   // DB2444
// stored: AutoNumber true, DBAccessibleFromOPCUA true, DBAccessibleFromWebserver true, InstanceOfName BoolToUDInt_Inverted_Filtered, InstanceOfType FB
"BoolToUDInt_Inverted_Filtered "
BEGIN
END_DATA_BLOCK

DATA_BLOCK "S1.CABINET061.ALARM2"   // DB2445
// stored: AutoNumber true, DBAccessibleFromOPCUA true, DBAccessibleFromWebserver true, InstanceOfName BoolToUDInt_Inverted_Filtered, InstanceOfType FB
"BoolToUDInt_Inverted_Filtered "
BEGIN
END_DATA_BLOCK

DATA_BLOCK "S1.CABINET061.WARNING1"   // DB2446
// stored: AutoNumber true, DBAccessibleFromOPCUA true, DBAccessibleFromWebserver true, InstanceOfName BoolToUDInt_Inverted_Filtered, InstanceOfType FB
"BoolToUDInt_Inverted_Filtered "
BEGIN
END_DATA_BLOCK

DATA_BLOCK "S1.CABINET061.WARNING2"   // DB2447
// stored: AutoNumber true, DBAccessibleFromOPCUA true, DBAccessibleFromWebserver true, InstanceOfName BoolToUDInt_Inverted_Filtered, InstanceOfType FB
"BoolToUDInt_Inverted_Filtered "
BEGIN
END_DATA_BLOCK

DATA_BLOCK "S1.CABINET062.ALARM1"   // DB2448
// stored: AutoNumber true, DBAccessibleFromOPCUA true, DBAccessibleFromWebserver true, InstanceOfName BoolToUDInt_Inverted_Filtered, InstanceOfType FB
"BoolToUDInt_Inverted_Filtered "
BEGIN
END_DATA_BLOCK

DATA_BLOCK "S1.CABINET062.ALARM2"   // DB2449
// stored: AutoNumber true, DBAccessibleFromOPCUA true, DBAccessibleFromWebserver true, InstanceOfName BoolToUDInt_Inverted_Filtered, InstanceOfType FB
"BoolToUDInt_Inverted_Filtered "
BEGIN
END_DATA_BLOCK

DATA_BLOCK "S1.CABINET062.WARNING1"   // DB2450
// stored: AutoNumber true, DBAccessibleFromOPCUA true, DBAccessibleFromWebserver true, InstanceOfName BoolToUDInt_Inverted_Filtered, InstanceOfType FB
"BoolToUDInt_Inverted_Filtered "
BEGIN
END_DATA_BLOCK

DATA_BLOCK "S1.CABINET062.WARNING2"   // DB2451
// stored: AutoNumber true, DBAccessibleFromOPCUA true, DBAccessibleFromWebserver true, InstanceOfName BoolToUDInt_Inverted_Filtered, InstanceOfType FB
"BoolToUDInt_Inverted_Filtered "
BEGIN
END_DATA_BLOCK

DATA_BLOCK "S1.CABINET063.ALARM1"   // DB2452
// stored: AutoNumber true, DBAccessibleFromOPCUA true, DBAccessibleFromWebserver true, InstanceOfName BoolToUDInt_Inverted_Filtered, InstanceOfType FB
"BoolToUDInt_Inverted_Filtered "
BEGIN
END_DATA_BLOCK

DATA_BLOCK "S1.CABINET063.ALARM2"   // DB2453
// stored: AutoNumber true, DBAccessibleFromOPCUA true, DBAccessibleFromWebserver true, InstanceOfName BoolToUDInt_Inverted_Filtered, InstanceOfType FB
"BoolToUDInt_Inverted_Filtered "
BEGIN
END_DATA_BLOCK

DATA_BLOCK "S1.CABINET063.WARNING1"   // DB2454
// stored: AutoNumber true, DBAccessibleFromOPCUA true, DBAccessibleFromWebserver true, InstanceOfName BoolToUDInt_Inverted_Filtered, InstanceOfType FB
"BoolToUDInt_Inverted_Filtered "
BEGIN
END_DATA_BLOCK

DATA_BLOCK "S1.CABINET063.WARNING2"   // DB2455
// stored: AutoNumber true, DBAccessibleFromOPCUA true, DBAccessibleFromWebserver true, InstanceOfName BoolToUDInt_Inverted_Filtered, InstanceOfType FB
"BoolToUDInt_Inverted_Filtered "
BEGIN
END_DATA_BLOCK

DATA_BLOCK "S1.CABINET064.ALARM1"   // DB2456
// stored: AutoNumber true, DBAccessibleFromOPCUA true, DBAccessibleFromWebserver true, InstanceOfName BoolToUDInt_Inverted_Filtered, InstanceOfType FB
"BoolToUDInt_Inverted_Filtered "
BEGIN
END_DATA_BLOCK

DATA_BLOCK "S1.CABINET064.ALARM2"   // DB2457
// stored: AutoNumber true, DBAccessibleFromOPCUA true, DBAccessibleFromWebserver true, InstanceOfName BoolToUDInt_Inverted_Filtered, InstanceOfType FB
"BoolToUDInt_Inverted_Filtered "
BEGIN
END_DATA_BLOCK

DATA_BLOCK "S1.CABINET064.WARNING1"   // DB2458
// stored: AutoNumber true, DBAccessibleFromOPCUA true, DBAccessibleFromWebserver true, InstanceOfName BoolToUDInt_Inverted_Filtered, InstanceOfType FB
"BoolToUDInt_Inverted_Filtered "
BEGIN
END_DATA_BLOCK

DATA_BLOCK "S1.CABINET064.WARNING2"   // DB2459
// stored: AutoNumber true, DBAccessibleFromOPCUA true, DBAccessibleFromWebserver true, InstanceOfName BoolToUDInt_Inverted_Filtered, InstanceOfType FB
"BoolToUDInt_Inverted_Filtered "
BEGIN
END_DATA_BLOCK

DATA_BLOCK "S1.CABINET065.ALARM1"   // DB2460
// stored: AutoNumber true, DBAccessibleFromOPCUA true, DBAccessibleFromWebserver true, InstanceOfName BoolToUDInt_Inverted_Filtered, InstanceOfType FB
"BoolToUDInt_Inverted_Filtered "
BEGIN
END_DATA_BLOCK

DATA_BLOCK "S1.CABINET065.ALARM2"   // DB2461
// stored: AutoNumber true, DBAccessibleFromOPCUA true, DBAccessibleFromWebserver true, InstanceOfName BoolToUDInt_Inverted_Filtered, InstanceOfType FB
"BoolToUDInt_Inverted_Filtered "
BEGIN
END_DATA_BLOCK

DATA_BLOCK "S1.CABINET065.WARNING1"   // DB2462
// stored: AutoNumber true, DBAccessibleFromOPCUA true, DBAccessibleFromWebserver true, InstanceOfName BoolToUDInt_Inverted_Filtered, InstanceOfType FB
"BoolToUDInt_Inverted_Filtered "
BEGIN
END_DATA_BLOCK

DATA_BLOCK "S1.CABINET065.WARNING2"   // DB2463
// stored: AutoNumber true, DBAccessibleFromOPCUA true, DBAccessibleFromWebserver true, InstanceOfName BoolToUDInt_Inverted_Filtered, InstanceOfType FB
"BoolToUDInt_Inverted_Filtered "
BEGIN
END_DATA_BLOCK

DATA_BLOCK "S1.CABINET066.ALARM1"   // DB2464
// stored: AutoNumber true, DBAccessibleFromOPCUA true, DBAccessibleFromWebserver true, InstanceOfName BoolToUDInt_Inverted_Filtered, InstanceOfType FB
"BoolToUDInt_Inverted_Filtered "
BEGIN
END_DATA_BLOCK

DATA_BLOCK "S1.CABINET066.ALARM2"   // DB2465
// stored: AutoNumber true, DBAccessibleFromOPCUA true, DBAccessibleFromWebserver true, InstanceOfName BoolToUDInt_Inverted_Filtered, InstanceOfType FB
"BoolToUDInt_Inverted_Filtered "
BEGIN
END_DATA_BLOCK

DATA_BLOCK "S1.CABINET066.WARNING1"   // DB2466
// stored: AutoNumber true, DBAccessibleFromOPCUA true, DBAccessibleFromWebserver true, InstanceOfName BoolToUDInt_Inverted_Filtered, InstanceOfType FB
"BoolToUDInt_Inverted_Filtered "
BEGIN
END_DATA_BLOCK

DATA_BLOCK "S1.CABINET066.WARNING2"   // DB2467
// stored: AutoNumber true, DBAccessibleFromOPCUA true, DBAccessibleFromWebserver true, InstanceOfName BoolToUDInt_Inverted_Filtered, InstanceOfType FB
"BoolToUDInt_Inverted_Filtered "
BEGIN
END_DATA_BLOCK

DATA_BLOCK "S1.CABINET067.ALARM1"   // DB2468
// stored: AutoNumber true, DBAccessibleFromOPCUA true, DBAccessibleFromWebserver true, InstanceOfName BoolToUDInt_Inverted_Filtered, InstanceOfType FB
"BoolToUDInt_Inverted_Filtered "
BEGIN
END_DATA_BLOCK

DATA_BLOCK "S1.CABINET067.ALARM2"   // DB2469
// stored: AutoNumber true, DBAccessibleFromOPCUA true, DBAccessibleFromWebserver true, InstanceOfName BoolToUDInt_Inverted_Filtered, InstanceOfType FB
"BoolToUDInt_Inverted_Filtered "
BEGIN
END_DATA_BLOCK

DATA_BLOCK "S1.CABINET067.WARNING1"   // DB2470
// stored: AutoNumber true, DBAccessibleFromOPCUA true, DBAccessibleFromWebserver true, InstanceOfName BoolToUDInt_Inverted_Filtered, InstanceOfType FB
"BoolToUDInt_Inverted_Filtered "
BEGIN
END_DATA_BLOCK

DATA_BLOCK "S1.CABINET067.WARNING2"   // DB2471
// stored: AutoNumber true, DBAccessibleFromOPCUA true, DBAccessibleFromWebserver true, InstanceOfName BoolToUDInt_Inverted_Filtered, InstanceOfType FB
"BoolToUDInt_Inverted_Filtered "
BEGIN
END_DATA_BLOCK

DATA_BLOCK "S1.CABINET068.ALARM1"   // DB2472
// stored: AutoNumber true, DBAccessibleFromOPCUA true, DBAccessibleFromWebserver true, InstanceOfName BoolToUDInt_Inverted_Filtered, InstanceOfType FB
"BoolToUDInt_Inverted_Filtered "
BEGIN
END_DATA_BLOCK

DATA_BLOCK "S1.CABINET068.ALARM2"   // DB2473
// stored: AutoNumber true, DBAccessibleFromOPCUA true, DBAccessibleFromWebserver true, InstanceOfName BoolToUDInt_Inverted_Filtered, InstanceOfType FB
"BoolToUDInt_Inverted_Filtered "
BEGIN
END_DATA_BLOCK

DATA_BLOCK "S1.CABINET068.WARNING1"   // DB2474
// stored: AutoNumber true, DBAccessibleFromOPCUA true, DBAccessibleFromWebserver true, InstanceOfName BoolToUDInt_Inverted_Filtered, InstanceOfType FB
"BoolToUDInt_Inverted_Filtered "
BEGIN
END_DATA_BLOCK

DATA_BLOCK "S1.CABINET068.WARNING2"   // DB2475
// stored: AutoNumber true, DBAccessibleFromOPCUA true, DBAccessibleFromWebserver true, InstanceOfName BoolToUDInt_Inverted_Filtered, InstanceOfType FB
"BoolToUDInt_Inverted_Filtered "
BEGIN
END_DATA_BLOCK

DATA_BLOCK "S1.CABINET069.ALARM1"   // DB2476
// stored: AutoNumber true, DBAccessibleFromOPCUA true, DBAccessibleFromWebserver true, InstanceOfName BoolToUDInt_Inverted_Filtered, InstanceOfType FB
"BoolToUDInt_Inverted_Filtered "
BEGIN
END_DATA_BLOCK

DATA_BLOCK "S1.CABINET069.ALARM2"   // DB2477
// stored: AutoNumber true, DBAccessibleFromOPCUA true, DBAccessibleFromWebserver true, InstanceOfName BoolToUDInt_Inverted_Filtered, InstanceOfType FB
"BoolToUDInt_Inverted_Filtered "
BEGIN
END_DATA_BLOCK

DATA_BLOCK "S1.CABINET069.WARNING1"   // DB2478
// stored: AutoNumber true, DBAccessibleFromOPCUA true, DBAccessibleFromWebserver true, InstanceOfName BoolToUDInt_Inverted_Filtered, InstanceOfType FB
"BoolToUDInt_Inverted_Filtered "
BEGIN
END_DATA_BLOCK

DATA_BLOCK "S1.CABINET069.WARNING2"   // DB2479
// stored: AutoNumber true, DBAccessibleFromOPCUA true, DBAccessibleFromWebserver true, InstanceOfName BoolToUDInt_Inverted_Filtered, InstanceOfType FB
"BoolToUDInt_Inverted_Filtered "
BEGIN
END_DATA_BLOCK

DATA_BLOCK "S1.CABINET070.ALARM1"   // DB2480
// stored: AutoNumber true, DBAccessibleFromOPCUA true, DBAccessibleFromWebserver true, InstanceOfName BoolToUDInt_Inverted_Filtered, InstanceOfType FB
"BoolToUDInt_Inverted_Filtered "
BEGIN
END_DATA_BLOCK

DATA_BLOCK "S1.CABINET070.ALARM2"   // DB2481
// stored: AutoNumber true, DBAccessibleFromOPCUA true, DBAccessibleFromWebserver true, InstanceOfName BoolToUDInt_Inverted_Filtered, InstanceOfType FB
"BoolToUDInt_Inverted_Filtered "
BEGIN
END_DATA_BLOCK

DATA_BLOCK "S1.CABINET070.WARNING1"   // DB2482
// stored: AutoNumber true, DBAccessibleFromOPCUA true, DBAccessibleFromWebserver true, InstanceOfName BoolToUDInt_Inverted_Filtered, InstanceOfType FB
"BoolToUDInt_Inverted_Filtered "
BEGIN
END_DATA_BLOCK

DATA_BLOCK "S1.CABINET070.WARNING2"   // DB2483
// stored: AutoNumber true, DBAccessibleFromOPCUA true, DBAccessibleFromWebserver true, InstanceOfName BoolToUDInt_Inverted_Filtered, InstanceOfType FB
"BoolToUDInt_Inverted_Filtered "
BEGIN
END_DATA_BLOCK

DATA_BLOCK "S1.CABINET071.ALARM1"   // DB2484
// stored: AutoNumber true, DBAccessibleFromOPCUA true, DBAccessibleFromWebserver true, InstanceOfName BoolToUDInt_Inverted_Filtered, InstanceOfType FB
"BoolToUDInt_Inverted_Filtered "
BEGIN
END_DATA_BLOCK

DATA_BLOCK "S1.CABINET071.ALARM2"   // DB2485
// stored: AutoNumber true, DBAccessibleFromOPCUA true, DBAccessibleFromWebserver true, InstanceOfName BoolToUDInt_Inverted_Filtered, InstanceOfType FB
"BoolToUDInt_Inverted_Filtered "
BEGIN
END_DATA_BLOCK

DATA_BLOCK "S1.CABINET071.WARNING1"   // DB2486
// stored: AutoNumber true, DBAccessibleFromOPCUA true, DBAccessibleFromWebserver true, InstanceOfName BoolToUDInt_Inverted_Filtered, InstanceOfType FB
"BoolToUDInt_Inverted_Filtered "
BEGIN
END_DATA_BLOCK

DATA_BLOCK "S1.CABINET071.WARNING2"   // DB2487
// stored: AutoNumber true, DBAccessibleFromOPCUA true, DBAccessibleFromWebserver true, InstanceOfName BoolToUDInt_Inverted_Filtered, InstanceOfType FB
"BoolToUDInt_Inverted_Filtered "
BEGIN
END_DATA_BLOCK

DATA_BLOCK "S1.CABINET072.ALARM1"   // DB2488
// stored: AutoNumber true, DBAccessibleFromOPCUA true, DBAccessibleFromWebserver true, InstanceOfName BoolToUDInt_Inverted_Filtered, InstanceOfType FB
"BoolToUDInt_Inverted_Filtered "
BEGIN
END_DATA_BLOCK

DATA_BLOCK "S1.CABINET072.ALARM2"   // DB2489
// stored: AutoNumber true, DBAccessibleFromOPCUA true, DBAccessibleFromWebserver true, InstanceOfName BoolToUDInt_Inverted_Filtered, InstanceOfType FB
"BoolToUDInt_Inverted_Filtered "
BEGIN
END_DATA_BLOCK

DATA_BLOCK "S1.CABINET072.WARNING1"   // DB2490
// stored: AutoNumber true, DBAccessibleFromOPCUA true, DBAccessibleFromWebserver true, InstanceOfName BoolToUDInt_Inverted_Filtered, InstanceOfType FB
"BoolToUDInt_Inverted_Filtered "
BEGIN
END_DATA_BLOCK

DATA_BLOCK "S1.CABINET072.WARNING2"   // DB2491
// stored: AutoNumber true, DBAccessibleFromOPCUA true, DBAccessibleFromWebserver true, InstanceOfName BoolToUDInt_Inverted_Filtered, InstanceOfType FB
"BoolToUDInt_Inverted_Filtered "
BEGIN
END_DATA_BLOCK

DATA_BLOCK "S1.CABINET073.ALARM1"   // DB2492
// stored: AutoNumber true, DBAccessibleFromOPCUA true, DBAccessibleFromWebserver true, InstanceOfName BoolToUDInt_Inverted_Filtered, InstanceOfType FB
"BoolToUDInt_Inverted_Filtered "
BEGIN
END_DATA_BLOCK

DATA_BLOCK "S1.CABINET073.ALARM2"   // DB2493
// stored: AutoNumber true, DBAccessibleFromOPCUA true, DBAccessibleFromWebserver true, InstanceOfName BoolToUDInt_Inverted_Filtered, InstanceOfType FB
"BoolToUDInt_Inverted_Filtered "
BEGIN
END_DATA_BLOCK

DATA_BLOCK "S1.CABINET073.WARNING1"   // DB2494
// stored: AutoNumber true, DBAccessibleFromOPCUA true, DBAccessibleFromWebserver true, InstanceOfName BoolToUDInt_Inverted_Filtered, InstanceOfType FB
"BoolToUDInt_Inverted_Filtered "
BEGIN
END_DATA_BLOCK

DATA_BLOCK "S1.CABINET073.WARNING2"   // DB2495
// stored: AutoNumber true, DBAccessibleFromOPCUA true, DBAccessibleFromWebserver true, InstanceOfName BoolToUDInt_Inverted_Filtered, InstanceOfType FB
"BoolToUDInt_Inverted_Filtered "
BEGIN
END_DATA_BLOCK

DATA_BLOCK "S1.CABINET074.ALARM1"   // DB2496
// stored: AutoNumber true, DBAccessibleFromOPCUA true, DBAccessibleFromWebserver true, InstanceOfName BoolToUDInt_Inverted_Filtered, InstanceOfType FB
"BoolToUDInt_Inverted_Filtered "
BEGIN
END_DATA_BLOCK

DATA_BLOCK "S1.CABINET074.ALARM2"   // DB2497
// stored: AutoNumber true, DBAccessibleFromOPCUA true, DBAccessibleFromWebserver true, InstanceOfName BoolToUDInt_Inverted_Filtered, InstanceOfType FB
"BoolToUDInt_Inverted_Filtered "
BEGIN
END_DATA_BLOCK

DATA_BLOCK "S1.CABINET074.WARNING1"   // DB2498
// stored: AutoNumber true, DBAccessibleFromOPCUA true, DBAccessibleFromWebserver true, InstanceOfName BoolToUDInt_Inverted_Filtered, InstanceOfType FB
"BoolToUDInt_Inverted_Filtered "
BEGIN
END_DATA_BLOCK

DATA_BLOCK "S1.CABINET074.WARNING2"   // DB2499
// stored: AutoNumber true, DBAccessibleFromOPCUA true, DBAccessibleFromWebserver true, InstanceOfName BoolToUDInt_Inverted_Filtered, InstanceOfType FB
"BoolToUDInt_Inverted_Filtered "
BEGIN
END_DATA_BLOCK

DATA_BLOCK "S1.CABINET075.ALARM1"   // DB2500
// stored: AutoNumber true, DBAccessibleFromOPCUA true, DBAccessibleFromWebserver true, InstanceOfName BoolToUDInt_Inverted_Filtered, InstanceOfType FB
"BoolToUDInt_Inverted_Filtered "
BEGIN
END_DATA_BLOCK

DATA_BLOCK "S1.CABINET075.ALARM2"   // DB2501
// stored: AutoNumber true, DBAccessibleFromOPCUA true, DBAccessibleFromWebserver true, InstanceOfName BoolToUDInt_Inverted_Filtered, InstanceOfType FB
"BoolToUDInt_Inverted_Filtered "
BEGIN
END_DATA_BLOCK

DATA_BLOCK "S1.CABINET075.WARNING1"   // DB2502
// stored: AutoNumber true, DBAccessibleFromOPCUA true, DBAccessibleFromWebserver true, InstanceOfName BoolToUDInt_Inverted_Filtered, InstanceOfType FB
"BoolToUDInt_Inverted_Filtered "
BEGIN
END_DATA_BLOCK

DATA_BLOCK "S1.CABINET075.WARNING2"   // DB2503
// stored: AutoNumber true, DBAccessibleFromOPCUA true, DBAccessibleFromWebserver true, InstanceOfName BoolToUDInt_Inverted_Filtered, InstanceOfType FB
"BoolToUDInt_Inverted_Filtered "
BEGIN
END_DATA_BLOCK

DATA_BLOCK "S1.CABINET076.ALARM1"   // DB2504
// stored: AutoNumber true, DBAccessibleFromOPCUA true, DBAccessibleFromWebserver true, InstanceOfName BoolToUDInt_Inverted_Filtered, InstanceOfType FB
"BoolToUDInt_Inverted_Filtered "
BEGIN
END_DATA_BLOCK

DATA_BLOCK "S1.CABINET076.ALARM2"   // DB2505
// stored: AutoNumber true, DBAccessibleFromOPCUA true, DBAccessibleFromWebserver true, InstanceOfName BoolToUDInt_Inverted_Filtered, InstanceOfType FB
"BoolToUDInt_Inverted_Filtered "
BEGIN
END_DATA_BLOCK

DATA_BLOCK "S1.CABINET076.WARNING1"   // DB2506
// stored: AutoNumber true, DBAccessibleFromOPCUA true, DBAccessibleFromWebserver true, InstanceOfName BoolToUDInt_Inverted_Filtered, InstanceOfType FB
"BoolToUDInt_Inverted_Filtered "
BEGIN
END_DATA_BLOCK

DATA_BLOCK "S1.CABINET076.WARNING2"   // DB2507
// stored: AutoNumber true, DBAccessibleFromOPCUA true, DBAccessibleFromWebserver true, InstanceOfName BoolToUDInt_Inverted_Filtered, InstanceOfType FB
"BoolToUDInt_Inverted_Filtered "
BEGIN
END_DATA_BLOCK

DATA_BLOCK "S1.CABINET077.ALARM1"   // DB2508
// stored: AutoNumber true, DBAccessibleFromOPCUA true, DBAccessibleFromWebserver true, InstanceOfName BoolToUDInt_Inverted_Filtered, InstanceOfType FB
"BoolToUDInt_Inverted_Filtered "
BEGIN
END_DATA_BLOCK

DATA_BLOCK "S1.CABINET077.ALARM2"   // DB2509
// stored: AutoNumber true, DBAccessibleFromOPCUA true, DBAccessibleFromWebserver true, InstanceOfName BoolToUDInt_Inverted_Filtered, InstanceOfType FB
"BoolToUDInt_Inverted_Filtered "
BEGIN
END_DATA_BLOCK

DATA_BLOCK "S1.CABINET077.WARNING1"   // DB2510
// stored: AutoNumber true, DBAccessibleFromOPCUA true, DBAccessibleFromWebserver true, InstanceOfName BoolToUDInt_Inverted_Filtered, InstanceOfType FB
"BoolToUDInt_Inverted_Filtered "
BEGIN
END_DATA_BLOCK

DATA_BLOCK "S1.CABINET077.WARNING2"   // DB2511
// stored: AutoNumber true, DBAccessibleFromOPCUA true, DBAccessibleFromWebserver true, InstanceOfName BoolToUDInt_Inverted_Filtered, InstanceOfType FB
"BoolToUDInt_Inverted_Filtered "
BEGIN
END_DATA_BLOCK

DATA_BLOCK "S1.CABINET078.ALARM1"   // DB2512
// stored: AutoNumber true, DBAccessibleFromOPCUA true, DBAccessibleFromWebserver true, InstanceOfName BoolToUDInt_Inverted_Filtered, InstanceOfType FB
"BoolToUDInt_Inverted_Filtered "
BEGIN
END_DATA_BLOCK

DATA_BLOCK "S1.CABINET078.ALARM2"   // DB2513
// stored: AutoNumber true, DBAccessibleFromOPCUA true, DBAccessibleFromWebserver true, InstanceOfName BoolToUDInt_Inverted_Filtered, InstanceOfType FB
"BoolToUDInt_Inverted_Filtered "
BEGIN
END_DATA_BLOCK

DATA_BLOCK "S1.CABINET078.WARNING1"   // DB2514
// stored: AutoNumber true, DBAccessibleFromOPCUA true, DBAccessibleFromWebserver true, InstanceOfName BoolToUDInt_Inverted_Filtered, InstanceOfType FB
"BoolToUDInt_Inverted_Filtered "
BEGIN
END_DATA_BLOCK

DATA_BLOCK "S1.CABINET078.WARNING2"   // DB2515
// stored: AutoNumber true, DBAccessibleFromOPCUA true, DBAccessibleFromWebserver true, InstanceOfName BoolToUDInt_Inverted_Filtered, InstanceOfType FB
"BoolToUDInt_Inverted_Filtered "
BEGIN
END_DATA_BLOCK

DATA_BLOCK "S1.CABINET079.ALARM1"   // DB2516
// stored: AutoNumber true, DBAccessibleFromOPCUA true, DBAccessibleFromWebserver true, InstanceOfName BoolToUDInt_Inverted_Filtered, InstanceOfType FB
"BoolToUDInt_Inverted_Filtered "
BEGIN
END_DATA_BLOCK

DATA_BLOCK "S1.CABINET079.ALARM2"   // DB2517
// stored: AutoNumber true, DBAccessibleFromOPCUA true, DBAccessibleFromWebserver true, InstanceOfName BoolToUDInt_Inverted_Filtered, InstanceOfType FB
"BoolToUDInt_Inverted_Filtered "
BEGIN
END_DATA_BLOCK

DATA_BLOCK "S1.CABINET079.WARNING1"   // DB2518
// stored: AutoNumber true, DBAccessibleFromOPCUA true, DBAccessibleFromWebserver true, InstanceOfName BoolToUDInt_Inverted_Filtered, InstanceOfType FB
"BoolToUDInt_Inverted_Filtered "
BEGIN
END_DATA_BLOCK

DATA_BLOCK "S1.CABINET079.WARNING2"   // DB2519
// stored: AutoNumber true, DBAccessibleFromOPCUA true, DBAccessibleFromWebserver true, InstanceOfName BoolToUDInt_Inverted_Filtered, InstanceOfType FB
"BoolToUDInt_Inverted_Filtered "
BEGIN
END_DATA_BLOCK

DATA_BLOCK "S1.CABINET080.ALARM1"   // DB2520
// stored: AutoNumber true, DBAccessibleFromOPCUA true, DBAccessibleFromWebserver true, InstanceOfName BoolToUDInt_Inverted_Filtered, InstanceOfType FB
"BoolToUDInt_Inverted_Filtered "
BEGIN
END_DATA_BLOCK

DATA_BLOCK "S1.CABINET080.ALARM2"   // DB2521
// stored: AutoNumber true, DBAccessibleFromOPCUA true, DBAccessibleFromWebserver true, InstanceOfName BoolToUDInt_Inverted_Filtered, InstanceOfType FB
"BoolToUDInt_Inverted_Filtered "
BEGIN
END_DATA_BLOCK

DATA_BLOCK "S1.CABINET080.WARNING1"   // DB2522
// stored: AutoNumber true, DBAccessibleFromOPCUA true, DBAccessibleFromWebserver true, InstanceOfName BoolToUDInt_Inverted_Filtered, InstanceOfType FB
"BoolToUDInt_Inverted_Filtered "
BEGIN
END_DATA_BLOCK

DATA_BLOCK "S1.CABINET080.WARNING2"   // DB2523
// stored: AutoNumber true, DBAccessibleFromOPCUA true, DBAccessibleFromWebserver true, InstanceOfName BoolToUDInt_Inverted_Filtered, InstanceOfType FB
"BoolToUDInt_Inverted_Filtered "
BEGIN
END_DATA_BLOCK

DATA_BLOCK "S1.CABINET081.ALARM1"   // DB2524
// stored: AutoNumber true, DBAccessibleFromOPCUA true, DBAccessibleFromWebserver true, InstanceOfName BoolToUDInt_Inverted_Filtered, InstanceOfType FB
"BoolToUDInt_Inverted_Filtered "
BEGIN
END_DATA_BLOCK

DATA_BLOCK "S1.CABINET081.ALARM2"   // DB2525
// stored: AutoNumber true, DBAccessibleFromOPCUA true, DBAccessibleFromWebserver true, InstanceOfName BoolToUDInt_Inverted_Filtered, InstanceOfType FB
"BoolToUDInt_Inverted_Filtered "
BEGIN
END_DATA_BLOCK

DATA_BLOCK "S1.CABINET081.WARNING1"   // DB2526
// stored: AutoNumber true, DBAccessibleFromOPCUA true, DBAccessibleFromWebserver true, InstanceOfName BoolToUDInt_Inverted_Filtered, InstanceOfType FB
"BoolToUDInt_Inverted_Filtered "
BEGIN
END_DATA_BLOCK

DATA_BLOCK "S1.CABINET081.WARNING2"   // DB2527
// stored: AutoNumber true, DBAccessibleFromOPCUA true, DBAccessibleFromWebserver true, InstanceOfName BoolToUDInt_Inverted_Filtered, InstanceOfType FB
"BoolToUDInt_Inverted_Filtered "
BEGIN
END_DATA_BLOCK

DATA_BLOCK "S1.CABINET082.ALARM1"   // DB2528
// stored: AutoNumber true, DBAccessibleFromOPCUA true, DBAccessibleFromWebserver true, InstanceOfName BoolToUDInt_Inverted_Filtered, InstanceOfType FB
"BoolToUDInt_Inverted_Filtered "
BEGIN
END_DATA_BLOCK

DATA_BLOCK "S1.CABINET082.ALARM2"   // DB2529
// stored: AutoNumber true, DBAccessibleFromOPCUA true, DBAccessibleFromWebserver true, InstanceOfName BoolToUDInt_Inverted_Filtered, InstanceOfType FB
"BoolToUDInt_Inverted_Filtered "
BEGIN
END_DATA_BLOCK

DATA_BLOCK "S1.CABINET082.WARNING1"   // DB2530
// stored: AutoNumber true, DBAccessibleFromOPCUA true, DBAccessibleFromWebserver true, InstanceOfName BoolToUDInt_Inverted_Filtered, InstanceOfType FB
"BoolToUDInt_Inverted_Filtered "
BEGIN
END_DATA_BLOCK

DATA_BLOCK "S1.CABINET082.WARNING2"   // DB2531
// stored: AutoNumber true, DBAccessibleFromOPCUA true, DBAccessibleFromWebserver true, InstanceOfName BoolToUDInt_Inverted_Filtered, InstanceOfType FB
"BoolToUDInt_Inverted_Filtered "
BEGIN
END_DATA_BLOCK

DATA_BLOCK "S1.CABINET083.ALARM1"   // DB2532
// stored: AutoNumber true, DBAccessibleFromOPCUA true, DBAccessibleFromWebserver true, InstanceOfName BoolToUDInt_Inverted_Filtered, InstanceOfType FB
"BoolToUDInt_Inverted_Filtered "
BEGIN
END_DATA_BLOCK

DATA_BLOCK "S1.CABINET083.ALARM2"   // DB2533
// stored: AutoNumber true, DBAccessibleFromOPCUA true, DBAccessibleFromWebserver true, InstanceOfName BoolToUDInt_Inverted_Filtered, InstanceOfType FB
"BoolToUDInt_Inverted_Filtered "
BEGIN
END_DATA_BLOCK

DATA_BLOCK "S1.CABINET083.WARNING1"   // DB2534
// stored: AutoNumber true, DBAccessibleFromOPCUA true, DBAccessibleFromWebserver true, InstanceOfName BoolToUDInt_Inverted_Filtered, InstanceOfType FB
"BoolToUDInt_Inverted_Filtered "
BEGIN
END_DATA_BLOCK

DATA_BLOCK "S1.CABINET083.WARNING2"   // DB2535
// stored: AutoNumber true, DBAccessibleFromOPCUA true, DBAccessibleFromWebserver true, InstanceOfName BoolToUDInt_Inverted_Filtered, InstanceOfType FB
"BoolToUDInt_Inverted_Filtered "
BEGIN
END_DATA_BLOCK

DATA_BLOCK "S1.CABINET084.ALARM1"   // DB2536
// stored: AutoNumber true, DBAccessibleFromOPCUA true, DBAccessibleFromWebserver true, InstanceOfName BoolToUDInt_Inverted_Filtered, InstanceOfType FB
"BoolToUDInt_Inverted_Filtered "
BEGIN
END_DATA_BLOCK

DATA_BLOCK "S1.CABINET084.ALARM2"   // DB2537
// stored: AutoNumber true, DBAccessibleFromOPCUA true, DBAccessibleFromWebserver true, InstanceOfName BoolToUDInt_Inverted_Filtered, InstanceOfType FB
"BoolToUDInt_Inverted_Filtered "
BEGIN
END_DATA_BLOCK

DATA_BLOCK "S1.CABINET084.WARNING1"   // DB2538
// stored: AutoNumber true, DBAccessibleFromOPCUA true, DBAccessibleFromWebserver true, InstanceOfName BoolToUDInt_Inverted_Filtered, InstanceOfType FB
"BoolToUDInt_Inverted_Filtered "
BEGIN
END_DATA_BLOCK

DATA_BLOCK "S1.CABINET084.WARNING2"   // DB2539
// stored: AutoNumber true, DBAccessibleFromOPCUA true, DBAccessibleFromWebserver true, InstanceOfName BoolToUDInt_Inverted_Filtered, InstanceOfType FB
"BoolToUDInt_Inverted_Filtered "
BEGIN
END_DATA_BLOCK

DATA_BLOCK "S1.CABINET085.ALARM1"   // DB2540
// stored: AutoNumber true, DBAccessibleFromOPCUA true, DBAccessibleFromWebserver true, InstanceOfName BoolToUDInt_Inverted_Filtered, InstanceOfType FB
"BoolToUDInt_Inverted_Filtered "
BEGIN
END_DATA_BLOCK

DATA_BLOCK "S1.CABINET085.ALARM2"   // DB2541
// stored: AutoNumber true, DBAccessibleFromOPCUA true, DBAccessibleFromWebserver true, InstanceOfName BoolToUDInt_Inverted_Filtered, InstanceOfType FB
"BoolToUDInt_Inverted_Filtered "
BEGIN
END_DATA_BLOCK

DATA_BLOCK "S1.CABINET085.WARNING1"   // DB2542
// stored: AutoNumber true, DBAccessibleFromOPCUA true, DBAccessibleFromWebserver true, InstanceOfName BoolToUDInt_Inverted_Filtered, InstanceOfType FB
"BoolToUDInt_Inverted_Filtered "
BEGIN
END_DATA_BLOCK

DATA_BLOCK "S1.CABINET085.WARNING2"   // DB2543
// stored: AutoNumber true, DBAccessibleFromOPCUA true, DBAccessibleFromWebserver true, InstanceOfName BoolToUDInt_Inverted_Filtered, InstanceOfType FB
"BoolToUDInt_Inverted_Filtered "
BEGIN
END_DATA_BLOCK

DATA_BLOCK "S1.CABINET086.ALARM1"   // DB2544
// stored: AutoNumber true, DBAccessibleFromOPCUA true, DBAccessibleFromWebserver true, InstanceOfName BoolToUDInt_Inverted_Filtered, InstanceOfType FB
"BoolToUDInt_Inverted_Filtered "
BEGIN
END_DATA_BLOCK

DATA_BLOCK "S1.CABINET086.ALARM2"   // DB2545
// stored: AutoNumber true, DBAccessibleFromOPCUA true, DBAccessibleFromWebserver true, InstanceOfName BoolToUDInt_Inverted_Filtered, InstanceOfType FB
"BoolToUDInt_Inverted_Filtered "
BEGIN
END_DATA_BLOCK

DATA_BLOCK "S1.CABINET086.WARNING1"   // DB2546
// stored: AutoNumber true, DBAccessibleFromOPCUA true, DBAccessibleFromWebserver true, InstanceOfName BoolToUDInt_Inverted_Filtered, InstanceOfType FB
"BoolToUDInt_Inverted_Filtered "
BEGIN
END_DATA_BLOCK

DATA_BLOCK "S1.CABINET086.WARNING2"   // DB2547
// stored: AutoNumber true, DBAccessibleFromOPCUA true, DBAccessibleFromWebserver true, InstanceOfName BoolToUDInt_Inverted_Filtered, InstanceOfType FB
"BoolToUDInt_Inverted_Filtered "
BEGIN
END_DATA_BLOCK

DATA_BLOCK "S1.CABINET087.ALARM1"   // DB2548
// stored: AutoNumber true, DBAccessibleFromOPCUA true, DBAccessibleFromWebserver true, InstanceOfName BoolToUDInt_Inverted_Filtered, InstanceOfType FB
"BoolToUDInt_Inverted_Filtered "
BEGIN
END_DATA_BLOCK

DATA_BLOCK "S1.CABINET087.ALARM2"   // DB2549
// stored: AutoNumber true, DBAccessibleFromOPCUA true, DBAccessibleFromWebserver true, InstanceOfName BoolToUDInt_Inverted_Filtered, InstanceOfType FB
"BoolToUDInt_Inverted_Filtered "
BEGIN
END_DATA_BLOCK

DATA_BLOCK "S1.CABINET087.WARNING1"   // DB2550
// stored: AutoNumber true, DBAccessibleFromOPCUA true, DBAccessibleFromWebserver true, InstanceOfName BoolToUDInt_Inverted_Filtered, InstanceOfType FB
"BoolToUDInt_Inverted_Filtered "
BEGIN
END_DATA_BLOCK

DATA_BLOCK "S1.CABINET087.WARNING2"   // DB2551
// stored: AutoNumber true, DBAccessibleFromOPCUA true, DBAccessibleFromWebserver true, InstanceOfName BoolToUDInt_Inverted_Filtered, InstanceOfType FB
"BoolToUDInt_Inverted_Filtered "
BEGIN
END_DATA_BLOCK

DATA_BLOCK "S1.CABINET088.ALARM1"   // DB2552
// stored: AutoNumber true, DBAccessibleFromOPCUA true, DBAccessibleFromWebserver true, InstanceOfName BoolToUDInt_Inverted_Filtered, InstanceOfType FB
"BoolToUDInt_Inverted_Filtered "
BEGIN
END_DATA_BLOCK

DATA_BLOCK "S1.CABINET088.ALARM2"   // DB2553
// stored: AutoNumber true, DBAccessibleFromOPCUA true, DBAccessibleFromWebserver true, InstanceOfName BoolToUDInt_Inverted_Filtered, InstanceOfType FB
"BoolToUDInt_Inverted_Filtered "
BEGIN
END_DATA_BLOCK

DATA_BLOCK "S1.CABINET088.WARNING1"   // DB2554
// stored: AutoNumber true, DBAccessibleFromOPCUA true, DBAccessibleFromWebserver true, InstanceOfName BoolToUDInt_Inverted_Filtered, InstanceOfType FB
"BoolToUDInt_Inverted_Filtered "
BEGIN
END_DATA_BLOCK

DATA_BLOCK "S1.CABINET088.WARNING2"   // DB2555
// stored: AutoNumber true, DBAccessibleFromOPCUA true, DBAccessibleFromWebserver true, InstanceOfName BoolToUDInt_Inverted_Filtered, InstanceOfType FB
"BoolToUDInt_Inverted_Filtered "
BEGIN
END_DATA_BLOCK

DATA_BLOCK "S1.CABINET089.ALARM1"   // DB2556
// stored: AutoNumber true, DBAccessibleFromOPCUA true, DBAccessibleFromWebserver true, InstanceOfName BoolToUDInt_Inverted_Filtered, InstanceOfType FB
"BoolToUDInt_Inverted_Filtered "
BEGIN
END_DATA_BLOCK

DATA_BLOCK "S1.CABINET089.ALARM2"   // DB2557
// stored: AutoNumber true, DBAccessibleFromOPCUA true, DBAccessibleFromWebserver true, InstanceOfName BoolToUDInt_Inverted_Filtered, InstanceOfType FB
"BoolToUDInt_Inverted_Filtered "
BEGIN
END_DATA_BLOCK

DATA_BLOCK "S1.CABINET089.WARNING1"   // DB2558
// stored: AutoNumber true, DBAccessibleFromOPCUA true, DBAccessibleFromWebserver true, InstanceOfName BoolToUDInt_Inverted_Filtered, InstanceOfType FB
"BoolToUDInt_Inverted_Filtered "
BEGIN
END_DATA_BLOCK

DATA_BLOCK "S1.CABINET089.WARNING2"   // DB2559
// stored: AutoNumber true, DBAccessibleFromOPCUA true, DBAccessibleFromWebserver true, InstanceOfName BoolToUDInt_Inverted_Filtered, InstanceOfType FB
"BoolToUDInt_Inverted_Filtered "
BEGIN
END_DATA_BLOCK

DATA_BLOCK "S1.CABINET090.ALARM1"   // DB2560
// stored: AutoNumber true, DBAccessibleFromOPCUA true, DBAccessibleFromWebserver true, InstanceOfName BoolToUDInt_Inverted_Filtered, InstanceOfType FB
"BoolToUDInt_Inverted_Filtered "
BEGIN
END_DATA_BLOCK

DATA_BLOCK "S1.CABINET090.ALARM2"   // DB2561
// stored: AutoNumber true, DBAccessibleFromOPCUA true, DBAccessibleFromWebserver true, InstanceOfName BoolToUDInt_Inverted_Filtered, InstanceOfType FB
"BoolToUDInt_Inverted_Filtered "
BEGIN
END_DATA_BLOCK

DATA_BLOCK "S1.CABINET090.WARNING1"   // DB2562
// stored: AutoNumber true, DBAccessibleFromOPCUA true, DBAccessibleFromWebserver true, InstanceOfName BoolToUDInt_Inverted_Filtered, InstanceOfType FB
"BoolToUDInt_Inverted_Filtered "
BEGIN
END_DATA_BLOCK

DATA_BLOCK "S1.CABINET090.WARNING2"   // DB2563
// stored: AutoNumber true, DBAccessibleFromOPCUA true, DBAccessibleFromWebserver true, InstanceOfName BoolToUDInt_Inverted_Filtered, InstanceOfType FB
"BoolToUDInt_Inverted_Filtered "
BEGIN
END_DATA_BLOCK

DATA_BLOCK "S1.CABINET091.ALARM1"   // DB2564
// stored: AutoNumber true, DBAccessibleFromOPCUA true, DBAccessibleFromWebserver true, InstanceOfName BoolToUDInt_Inverted_Filtered, InstanceOfType FB
"BoolToUDInt_Inverted_Filtered "
BEGIN
END_DATA_BLOCK

DATA_BLOCK "S1.CABINET091.ALARM2"   // DB2565
// stored: AutoNumber true, DBAccessibleFromOPCUA true, DBAccessibleFromWebserver true, InstanceOfName BoolToUDInt_Inverted_Filtered, InstanceOfType FB
"BoolToUDInt_Inverted_Filtered "
BEGIN
END_DATA_BLOCK

DATA_BLOCK "S1.CABINET091.WARNING1"   // DB2566
// stored: AutoNumber true, DBAccessibleFromOPCUA true, DBAccessibleFromWebserver true, InstanceOfName BoolToUDInt_Inverted_Filtered, InstanceOfType FB
"BoolToUDInt_Inverted_Filtered "
BEGIN
END_DATA_BLOCK

DATA_BLOCK "S1.CABINET091.WARNING2"   // DB2567
// stored: AutoNumber true, DBAccessibleFromOPCUA true, DBAccessibleFromWebserver true, InstanceOfName BoolToUDInt_Inverted_Filtered, InstanceOfType FB
"BoolToUDInt_Inverted_Filtered "
BEGIN
END_DATA_BLOCK

DATA_BLOCK "S1.CABINET092.ALARM1"   // DB2568
// stored: AutoNumber true, DBAccessibleFromOPCUA true, DBAccessibleFromWebserver true, InstanceOfName BoolToUDInt_Inverted_Filtered, InstanceOfType FB
"BoolToUDInt_Inverted_Filtered "
BEGIN
END_DATA_BLOCK

DATA_BLOCK "S1.CABINET092.ALARM2"   // DB2569
// stored: AutoNumber true, DBAccessibleFromOPCUA true, DBAccessibleFromWebserver true, InstanceOfName BoolToUDInt_Inverted_Filtered, InstanceOfType FB
"BoolToUDInt_Inverted_Filtered "
BEGIN
END_DATA_BLOCK

DATA_BLOCK "S1.CABINET092.WARNING1"   // DB2570
// stored: AutoNumber true, DBAccessibleFromOPCUA true, DBAccessibleFromWebserver true, InstanceOfName BoolToUDInt_Inverted_Filtered, InstanceOfType FB
"BoolToUDInt_Inverted_Filtered "
BEGIN
END_DATA_BLOCK

DATA_BLOCK "S1.CABINET092.WARNING2"   // DB2571
// stored: AutoNumber true, DBAccessibleFromOPCUA true, DBAccessibleFromWebserver true, InstanceOfName BoolToUDInt_Inverted_Filtered, InstanceOfType FB
"BoolToUDInt_Inverted_Filtered "
BEGIN
END_DATA_BLOCK

DATA_BLOCK "S1.CABINET093.ALARM1"   // DB2572
// stored: AutoNumber true, DBAccessibleFromOPCUA true, DBAccessibleFromWebserver true, InstanceOfName BoolToUDInt_Inverted_Filtered, InstanceOfType FB
"BoolToUDInt_Inverted_Filtered "
BEGIN
END_DATA_BLOCK

DATA_BLOCK "S1.CABINET093.ALARM2"   // DB2573
// stored: AutoNumber true, DBAccessibleFromOPCUA true, DBAccessibleFromWebserver true, InstanceOfName BoolToUDInt_Inverted_Filtered, InstanceOfType FB
"BoolToUDInt_Inverted_Filtered "
BEGIN
END_DATA_BLOCK

DATA_BLOCK "S1.CABINET093.WARNING1"   // DB2574
// stored: AutoNumber true, DBAccessibleFromOPCUA true, DBAccessibleFromWebserver true, InstanceOfName BoolToUDInt_Inverted_Filtered, InstanceOfType FB
"BoolToUDInt_Inverted_Filtered "
BEGIN
END_DATA_BLOCK

DATA_BLOCK "S1.CABINET093.WARNING2"   // DB2575
// stored: AutoNumber true, DBAccessibleFromOPCUA true, DBAccessibleFromWebserver true, InstanceOfName BoolToUDInt_Inverted_Filtered, InstanceOfType FB
"BoolToUDInt_Inverted_Filtered "
BEGIN
END_DATA_BLOCK

DATA_BLOCK "S1.CABINET094.ALARM1"   // DB2576
// stored: AutoNumber true, DBAccessibleFromOPCUA true, DBAccessibleFromWebserver true, InstanceOfName BoolToUDInt_Inverted_Filtered, InstanceOfType FB
"BoolToUDInt_Inverted_Filtered "
BEGIN
END_DATA_BLOCK

DATA_BLOCK "S1.CABINET094.ALARM2"   // DB2577
// stored: AutoNumber true, DBAccessibleFromOPCUA true, DBAccessibleFromWebserver true, InstanceOfName BoolToUDInt_Inverted_Filtered, InstanceOfType FB
"BoolToUDInt_Inverted_Filtered "
BEGIN
END_DATA_BLOCK

DATA_BLOCK "S1.CABINET094.WARNING1"   // DB2578
// stored: AutoNumber true, DBAccessibleFromOPCUA true, DBAccessibleFromWebserver true, InstanceOfName BoolToUDInt_Inverted_Filtered, InstanceOfType FB
"BoolToUDInt_Inverted_Filtered "
BEGIN
END_DATA_BLOCK

DATA_BLOCK "S1.CABINET094.WARNING2"   // DB2579
// stored: AutoNumber true, DBAccessibleFromOPCUA true, DBAccessibleFromWebserver true, InstanceOfName BoolToUDInt_Inverted_Filtered, InstanceOfType FB
"BoolToUDInt_Inverted_Filtered "
BEGIN
END_DATA_BLOCK

DATA_BLOCK "S1.CABINET095.ALARM1"   // DB2580
// stored: AutoNumber true, DBAccessibleFromOPCUA true, DBAccessibleFromWebserver true, InstanceOfName BoolToUDInt_Inverted_Filtered, InstanceOfType FB
"BoolToUDInt_Inverted_Filtered "
BEGIN
END_DATA_BLOCK

DATA_BLOCK "S1.CABINET095.ALARM2"   // DB2581
// stored: AutoNumber true, DBAccessibleFromOPCUA true, DBAccessibleFromWebserver true, InstanceOfName BoolToUDInt_Inverted_Filtered, InstanceOfType FB
"BoolToUDInt_Inverted_Filtered "
BEGIN
END_DATA_BLOCK

DATA_BLOCK "S1.CABINET095.WARNING1"   // DB2582
// stored: AutoNumber true, DBAccessibleFromOPCUA true, DBAccessibleFromWebserver true, InstanceOfName BoolToUDInt_Inverted_Filtered, InstanceOfType FB
"BoolToUDInt_Inverted_Filtered "
BEGIN
END_DATA_BLOCK

DATA_BLOCK "S1.CABINET095.WARNING2"   // DB2583
// stored: AutoNumber true, DBAccessibleFromOPCUA true, DBAccessibleFromWebserver true, InstanceOfName BoolToUDInt_Inverted_Filtered, InstanceOfType FB
"BoolToUDInt_Inverted_Filtered "
BEGIN
END_DATA_BLOCK

DATA_BLOCK "S1.CABINET096.ALARM1"   // DB2584
// stored: AutoNumber true, DBAccessibleFromOPCUA true, DBAccessibleFromWebserver true, InstanceOfName BoolToUDInt_Inverted_Filtered, InstanceOfType FB
"BoolToUDInt_Inverted_Filtered "
BEGIN
END_DATA_BLOCK

DATA_BLOCK "S1.CABINET096.ALARM2"   // DB2585
// stored: AutoNumber true, DBAccessibleFromOPCUA true, DBAccessibleFromWebserver true, InstanceOfName BoolToUDInt_Inverted_Filtered, InstanceOfType FB
"BoolToUDInt_Inverted_Filtered "
BEGIN
END_DATA_BLOCK

DATA_BLOCK "S1.CABINET096.WARNING1"   // DB2586
// stored: AutoNumber true, DBAccessibleFromOPCUA true, DBAccessibleFromWebserver true, InstanceOfName BoolToUDInt_Inverted_Filtered, InstanceOfType FB
"BoolToUDInt_Inverted_Filtered "
BEGIN
END_DATA_BLOCK

DATA_BLOCK "S1.CABINET096.WARNING2"   // DB2587
// stored: AutoNumber true, DBAccessibleFromOPCUA true, DBAccessibleFromWebserver true, InstanceOfName BoolToUDInt_Inverted_Filtered, InstanceOfType FB
"BoolToUDInt_Inverted_Filtered "
BEGIN
END_DATA_BLOCK

DATA_BLOCK "S1.CABINET097.ALARM1"   // DB2588
// stored: AutoNumber true, DBAccessibleFromOPCUA true, DBAccessibleFromWebserver true, InstanceOfName BoolToUDInt_Inverted_Filtered, InstanceOfType FB
"BoolToUDInt_Inverted_Filtered "
BEGIN
END_DATA_BLOCK

